   HoldingRegisters[2603] := 16#0000;
   HoldingRegisters[2604] := 16#0000;
   HoldingRegisters[2605] := 16#0000;
   HoldingRegisters[2606] := 16#0000;
   HoldingRegisters[2607] := 16#0000;
   HoldingRegisters[2608] := 16#0000;
   HoldingRegisters[2609] := 16#0000;
   HoldingRegisters[2610] := 16#0000;
   HoldingRegisters[2611] := 16#0000;
   HoldingRegisters[2612] := 16#0000;
   HoldingRegisters[2613] := 16#0000;
   HoldingRegisters[2614] := 16#0000;
   HoldingRegisters[2615] := 16#0000;
   HoldingRegisters[2616] := 16#0000;
   HoldingRegisters[2617] := 16#0000;
   HoldingRegisters[2618] := 16#0000;
   HoldingRegisters[2619] := 16#0000;
   HoldingRegisters[2620] := 16#0000;
   HoldingRegisters[2621] := 16#0000;
   HoldingRegisters[2622] := 16#0000;
   HoldingRegisters[2623] := 16#0000;
   HoldingRegisters[2624] := 16#0000;
   HoldingRegisters[2625] := 16#0000;
   HoldingRegisters[2626] := 16#0000;
   HoldingRegisters[2627] := 16#0000;
   HoldingRegisters[2628] := 16#0000;
   HoldingRegisters[2629] := 16#0000;
   HoldingRegisters[2630] := 16#0000;
   HoldingRegisters[2631] := 16#0000;
   HoldingRegisters[2632] := 16#0000;
   HoldingRegisters[2633] := 16#0000;
   HoldingRegisters[2634] := 16#0000;
   HoldingRegisters[2635] := 16#0000;
   HoldingRegisters[2636] := 16#0000;
   HoldingRegisters[2637] := 16#0000;
   HoldingRegisters[2638] := 16#0000;
   HoldingRegisters[2639] := 16#0000;
   HoldingRegisters[2640] := 16#0000;
   HoldingRegisters[2641] := 16#0000;
   HoldingRegisters[2642] := 16#0000;
   HoldingRegisters[2643] := 16#0000;
   HoldingRegisters[2644] := 16#0000;
   HoldingRegisters[2645] := 16#0000;
   HoldingRegisters[2646] := 16#0000;
   HoldingRegisters[2647] := 16#0000;
   HoldingRegisters[2648] := 16#0000;
   HoldingRegisters[2649] := 16#0000;
   HoldingRegisters[2650] := 16#0000;
   HoldingRegisters[2651] := 16#0000;
   HoldingRegisters[2652] := 16#0000;
   HoldingRegisters[2653] := 16#0000;
   HoldingRegisters[2654] := 16#0000;
   HoldingRegisters[2655] := 16#0000;
   HoldingRegisters[2656] := 16#0000;
   HoldingRegisters[2657] := 16#0000;
   HoldingRegisters[2658] := 16#0000;
   HoldingRegisters[2659] := 16#0000;
   HoldingRegisters[2660] := 16#0000;
   HoldingRegisters[2661] := 16#0000;
   HoldingRegisters[2662] := 16#0000;
   HoldingRegisters[2663] := 16#0000;
   HoldingRegisters[2664] := 16#0000;
   HoldingRegisters[2665] := 16#0000;
   HoldingRegisters[2666] := 16#0000;
   HoldingRegisters[2667] := 16#0000;
   HoldingRegisters[2668] := 16#0000;
   HoldingRegisters[2669] := 16#0000;
   HoldingRegisters[2670] := 16#0000;
   HoldingRegisters[2671] := 16#0000;
   HoldingRegisters[2672] := 16#0000;
   HoldingRegisters[2673] := 16#0000;
   HoldingRegisters[2674] := 16#0000;
   HoldingRegisters[2675] := 16#0000;
   HoldingRegisters[2676] := 16#0000;
   HoldingRegisters[2677] := 16#0000;
   HoldingRegisters[2678] := 16#0000;
   HoldingRegisters[2679] := 16#0000;
   HoldingRegisters[2680] := 16#0000;
   HoldingRegisters[2681] := 16#0000;
   HoldingRegisters[2682] := 16#0000;
   HoldingRegisters[2683] := 16#0000;
   HoldingRegisters[2684] := 16#0000;
   HoldingRegisters[2685] := 16#0000;
   HoldingRegisters[2686] := 16#0000;
   HoldingRegisters[2687] := 16#0000;
   HoldingRegisters[2688] := 16#0000;
   HoldingRegisters[2689] := 16#0000;
   HoldingRegisters[2690] := 16#0000;
   HoldingRegisters[2691] := 16#0000;
   HoldingRegisters[2692] := 16#0000;
   HoldingRegisters[2693] := 16#0000;
   HoldingRegisters[2694] := 16#0000;
   HoldingRegisters[2695] := 16#0000;
   HoldingRegisters[2696] := 16#0000;
   HoldingRegisters[2697] := 16#0000;
   HoldingRegisters[2698] := 16#0000;
   HoldingRegisters[2699] := 16#0000;
   HoldingRegisters[2700] := 16#0000;
   HoldingRegisters[2701] := 16#0000;
   HoldingRegisters[2702] := 16#0000;
   HoldingRegisters[2703] := 16#0000;
   HoldingRegisters[2704] := 16#0000;
   HoldingRegisters[2705] := 16#0000;
   HoldingRegisters[2706] := 16#0000;
   HoldingRegisters[2707] := 16#0000;
   HoldingRegisters[2708] := 16#0000;
   HoldingRegisters[2709] := 16#0000;
   HoldingRegisters[2710] := 16#0000;
   HoldingRegisters[2711] := 16#0000;
   HoldingRegisters[2712] := 16#0000;
   HoldingRegisters[2713] := 16#0000;
   HoldingRegisters[2714] := 16#0000;
   HoldingRegisters[2715] := 16#0000;
   HoldingRegisters[2716] := 16#0000;
   HoldingRegisters[2717] := 16#0000;
   HoldingRegisters[2718] := 16#0000;
   HoldingRegisters[2719] := 16#0000;
   HoldingRegisters[2720] := 16#0000;
   HoldingRegisters[2721] := 16#0000;
   HoldingRegisters[2722] := 16#0000;
   HoldingRegisters[2723] := 16#0000;
   HoldingRegisters[2724] := 16#0000;
   HoldingRegisters[2725] := 16#0000;
   HoldingRegisters[2726] := 16#0000;
   HoldingRegisters[2727] := 16#0000;
   HoldingRegisters[2728] := 16#0000;
   HoldingRegisters[2729] := 16#0000;
   HoldingRegisters[2730] := 16#0000;
   HoldingRegisters[2731] := 16#0000;
   HoldingRegisters[2732] := 16#0000;
   HoldingRegisters[2733] := 16#0000;
   HoldingRegisters[2734] := 16#0000;
   HoldingRegisters[2735] := 16#0000;
   HoldingRegisters[2736] := 16#0000;
   HoldingRegisters[2737] := 16#0000;
   HoldingRegisters[2738] := 16#0000;
   HoldingRegisters[2739] := 16#0000;
   HoldingRegisters[2740] := 16#0000;
   HoldingRegisters[2741] := 16#0000;
   HoldingRegisters[2742] := 16#0000;
   HoldingRegisters[2743] := 16#0000;
   HoldingRegisters[2744] := 16#0000;
   HoldingRegisters[2745] := 16#0000;
   HoldingRegisters[2746] := 16#0000;
   HoldingRegisters[2747] := 16#0000;
   HoldingRegisters[2748] := 16#0000;
   HoldingRegisters[2749] := 16#0000;
   HoldingRegisters[2750] := 16#0000;
   HoldingRegisters[2751] := 16#0000;
   HoldingRegisters[2752] := 16#0000;
   HoldingRegisters[2753] := 16#0000;
   HoldingRegisters[2754] := 16#0000;
   HoldingRegisters[2755] := 16#0000;
   HoldingRegisters[2756] := 16#0000;
   HoldingRegisters[2757] := 16#0000;
   HoldingRegisters[2758] := 16#0000;
   HoldingRegisters[2759] := 16#0000;
   HoldingRegisters[2760] := 16#0000;
   HoldingRegisters[2761] := 16#0000;
   HoldingRegisters[2762] := 16#0000;
   HoldingRegisters[2763] := 16#0000;
   HoldingRegisters[2764] := 16#0000;
   HoldingRegisters[2765] := 16#0000;
   HoldingRegisters[2766] := 16#0000;
   HoldingRegisters[2767] := 16#0000;
   HoldingRegisters[2768] := 16#0000;
   HoldingRegisters[2769] := 16#0000;
   HoldingRegisters[2770] := 16#0000;
   HoldingRegisters[2771] := 16#0000;
   HoldingRegisters[2772] := 16#0000;
   HoldingRegisters[2773] := 16#0000;
   HoldingRegisters[2774] := 16#0000;
   HoldingRegisters[2775] := 16#0000;
   HoldingRegisters[2776] := 16#0000;
   HoldingRegisters[2777] := 16#0000;
   HoldingRegisters[2778] := 16#0000;
   HoldingRegisters[2779] := 16#0000;
   HoldingRegisters[2780] := 16#0000;
   HoldingRegisters[2781] := 16#0000;
   HoldingRegisters[2782] := 16#0000;
   HoldingRegisters[2783] := 16#0000;
   HoldingRegisters[2784] := 16#0000;
   HoldingRegisters[2785] := 16#0000;
   HoldingRegisters[2786] := 16#0000;
   HoldingRegisters[2787] := 16#0000;
   HoldingRegisters[2788] := 16#0000;
   HoldingRegisters[2789] := 16#0000;
   HoldingRegisters[2790] := 16#0000;
   HoldingRegisters[2791] := 16#0000;
   HoldingRegisters[2792] := 16#0000;
   HoldingRegisters[2793] := 16#0000;
   HoldingRegisters[2794] := 16#0000;
   HoldingRegisters[2795] := 16#0000;
   HoldingRegisters[2796] := 16#0000;
   HoldingRegisters[2797] := 16#0000;
   HoldingRegisters[2798] := 16#0000;
   HoldingRegisters[2799] := 16#0000;
   HoldingRegisters[2800] := 16#0000;
   HoldingRegisters[2801] := 16#0000;
   HoldingRegisters[2802] := 16#0000;
   HoldingRegisters[2803] := 16#0000;
   HoldingRegisters[2804] := 16#0000;
   HoldingRegisters[2805] := 16#0000;
   HoldingRegisters[2806] := 16#0000;
   HoldingRegisters[2807] := 16#0000;
   HoldingRegisters[2808] := 16#0000;
   HoldingRegisters[2809] := 16#0000;
   HoldingRegisters[2810] := 16#0000;
   HoldingRegisters[2811] := 16#0000;
   HoldingRegisters[2812] := 16#0000;
   HoldingRegisters[2813] := 16#0000;
   HoldingRegisters[2814] := 16#0000;
   HoldingRegisters[2815] := 16#0000;
   HoldingRegisters[2816] := 16#0000;
   HoldingRegisters[2817] := 16#0000;
   HoldingRegisters[2818] := 16#0000;
   HoldingRegisters[2819] := 16#0000;
   HoldingRegisters[2820] := 16#0000;
   HoldingRegisters[2821] := 16#0000;
   HoldingRegisters[2822] := 16#0000;
   HoldingRegisters[2823] := 16#0000;
   HoldingRegisters[2824] := 16#0000;
   HoldingRegisters[2825] := 16#0000;
   HoldingRegisters[2826] := 16#0000;
   HoldingRegisters[2827] := 16#0000;
   HoldingRegisters[2828] := 16#0000;
   HoldingRegisters[2829] := 16#0000;
   HoldingRegisters[2830] := 16#0000;
   HoldingRegisters[2831] := 16#0000;
   HoldingRegisters[2832] := 16#0000;
   HoldingRegisters[2833] := 16#0000;
   HoldingRegisters[2834] := 16#0000;
   HoldingRegisters[2835] := 16#0000;
   HoldingRegisters[2836] := 16#0000;
   HoldingRegisters[2837] := 16#0000;
   HoldingRegisters[2838] := 16#0000;
   HoldingRegisters[2839] := 16#0000;
   HoldingRegisters[2840] := 16#0000;
   HoldingRegisters[2841] := 16#0000;
   HoldingRegisters[2842] := 16#0000;
   HoldingRegisters[2843] := 16#0000;
   HoldingRegisters[2844] := 16#0000;
   HoldingRegisters[2845] := 16#0000;
   HoldingRegisters[2846] := 16#0000;
   HoldingRegisters[2847] := 16#0000;
   HoldingRegisters[2848] := 16#0000;
   HoldingRegisters[2849] := 16#0000;
   HoldingRegisters[2850] := 16#0000;
   HoldingRegisters[2851] := 16#0000;
   HoldingRegisters[2852] := 16#0000;
   HoldingRegisters[2853] := 16#0000;
   HoldingRegisters[2854] := 16#0000;
   HoldingRegisters[2855] := 16#0000;
   HoldingRegisters[2856] := 16#0000;
   HoldingRegisters[2857] := 16#0000;
   HoldingRegisters[2858] := 16#0000;
   HoldingRegisters[2859] := 16#0000;
   HoldingRegisters[2860] := 16#0000;
   HoldingRegisters[2861] := 16#0000;
   HoldingRegisters[2862] := 16#0000;
   HoldingRegisters[2863] := 16#0000;
   HoldingRegisters[2864] := 16#0000;
   HoldingRegisters[2865] := 16#0000;
   HoldingRegisters[2866] := 16#0000;
   HoldingRegisters[2867] := 16#0000;
   HoldingRegisters[2868] := 16#0000;
   HoldingRegisters[2869] := 16#0000;
   HoldingRegisters[2870] := 16#0000;
   HoldingRegisters[2871] := 16#0000;
   HoldingRegisters[2872] := 16#0000;
   HoldingRegisters[2873] := 16#0000;
   HoldingRegisters[2874] := 16#0000;
   HoldingRegisters[2875] := 16#0000;
   HoldingRegisters[2876] := 16#0000;
   HoldingRegisters[2877] := 16#0000;
   HoldingRegisters[2878] := 16#0000;
   HoldingRegisters[2879] := 16#0000;
   HoldingRegisters[2880] := 16#0000;
   HoldingRegisters[2881] := 16#0000;
   HoldingRegisters[2882] := 16#0000;
   HoldingRegisters[2883] := 16#0000;
   HoldingRegisters[2884] := 16#0000;
   HoldingRegisters[2885] := 16#0000;
   HoldingRegisters[2886] := 16#0000;
   HoldingRegisters[2887] := 16#0000;
   HoldingRegisters[2888] := 16#0000;
   HoldingRegisters[2889] := 16#0000;
   HoldingRegisters[2890] := 16#0000;
   HoldingRegisters[2891] := 16#0000;
   HoldingRegisters[2892] := 16#0000;
   HoldingRegisters[2893] := 16#0000;
   HoldingRegisters[2894] := 16#0000;
   HoldingRegisters[2895] := 16#0000;
   HoldingRegisters[2896] := 16#0000;
   HoldingRegisters[2897] := 16#0000;
   HoldingRegisters[2898] := 16#0000;
   HoldingRegisters[2899] := 16#0000;
   HoldingRegisters[2900] := 16#0000;
   HoldingRegisters[2901] := 16#0000;
   HoldingRegisters[2902] := 16#0000;
   HoldingRegisters[2903] := 16#0000;
   HoldingRegisters[2904] := 16#0000;
   HoldingRegisters[2905] := 16#0000;
   HoldingRegisters[2906] := 16#0000;
   HoldingRegisters[2907] := 16#0000;
   HoldingRegisters[2908] := 16#0000;
   HoldingRegisters[2909] := 16#0000;
   HoldingRegisters[2910] := 16#0000;
   HoldingRegisters[2911] := 16#0000;
   HoldingRegisters[2912] := 16#0000;
   HoldingRegisters[2913] := 16#0000;
   HoldingRegisters[2914] := 16#0000;
   HoldingRegisters[2915] := 16#0000;
   HoldingRegisters[2916] := 16#0000;
   HoldingRegisters[2917] := 16#0000;
   HoldingRegisters[2918] := 16#0000;
   HoldingRegisters[2919] := 16#0000;
   HoldingRegisters[2920] := 16#0000;
   HoldingRegisters[2921] := 16#0000;
   HoldingRegisters[2922] := 16#0000;
   HoldingRegisters[2923] := 16#0000;
   HoldingRegisters[2924] := 16#0000;
   HoldingRegisters[2925] := 16#0000;
   HoldingRegisters[2926] := 16#0000;
   HoldingRegisters[2927] := 16#0000;
   HoldingRegisters[2928] := 16#0000;
   HoldingRegisters[2929] := 16#0000;
   HoldingRegisters[2930] := 16#0000;
   HoldingRegisters[2931] := 16#0000;
   HoldingRegisters[2932] := 16#0000;
   HoldingRegisters[2933] := 16#0000;
   HoldingRegisters[2934] := 16#0000;
   HoldingRegisters[2935] := 16#0000;
   HoldingRegisters[2936] := 16#0000;
   HoldingRegisters[2937] := 16#0000;
   HoldingRegisters[2938] := 16#0000;
   HoldingRegisters[2939] := 16#0000;
   HoldingRegisters[2940] := 16#0000;
   HoldingRegisters[2941] := 16#0000;
   HoldingRegisters[2942] := 16#0000;
   HoldingRegisters[2943] := 16#0000;
   HoldingRegisters[2944] := 16#0000;
   HoldingRegisters[2945] := 16#0000;
   HoldingRegisters[2946] := 16#0000;
   HoldingRegisters[2947] := 16#0000;
   HoldingRegisters[2948] := 16#0000;
   HoldingRegisters[2949] := 16#0000;
   HoldingRegisters[2950] := 16#0000;
   HoldingRegisters[2951] := 16#0000;
   HoldingRegisters[2952] := 16#0000;
   HoldingRegisters[2953] := 16#0000;
   HoldingRegisters[2954] := 16#0000;
   HoldingRegisters[2955] := 16#0000;
   HoldingRegisters[2956] := 16#0000;
   HoldingRegisters[2957] := 16#0000;
   HoldingRegisters[2958] := 16#0000;
   HoldingRegisters[2959] := 16#0000;
   HoldingRegisters[2960] := 16#0000;
   HoldingRegisters[2961] := 16#0000;
   HoldingRegisters[2962] := 16#0000;
   HoldingRegisters[2963] := 16#0000;
   HoldingRegisters[2964] := 16#0000;
   HoldingRegisters[2965] := 16#0000;
   HoldingRegisters[2966] := 16#0000;
   HoldingRegisters[2967] := 16#0000;
   HoldingRegisters[2968] := 16#0000;
   HoldingRegisters[2969] := 16#0000;
   HoldingRegisters[2970] := 16#0000;
   HoldingRegisters[2971] := 16#0000;
   HoldingRegisters[2972] := 16#0000;
   HoldingRegisters[2973] := 16#0000;
   HoldingRegisters[2974] := 16#0000;
   HoldingRegisters[2975] := 16#0000;
   HoldingRegisters[2976] := 16#0000;
   HoldingRegisters[2977] := 16#0000;
   HoldingRegisters[2978] := 16#0000;
   HoldingRegisters[2979] := 16#0000;
   HoldingRegisters[2980] := 16#0000;
   HoldingRegisters[2981] := 16#0000;
   HoldingRegisters[2982] := 16#0000;
   HoldingRegisters[2983] := 16#0000;
   HoldingRegisters[2984] := 16#0000;
   HoldingRegisters[2985] := 16#0000;
   HoldingRegisters[2986] := 16#0000;
   HoldingRegisters[2987] := 16#0000;
   HoldingRegisters[2988] := 16#0000;
   HoldingRegisters[2989] := 16#0000;
   HoldingRegisters[2990] := 16#0000;
   HoldingRegisters[2991] := 16#0000;
   HoldingRegisters[2992] := 16#0000;
   HoldingRegisters[2993] := 16#0000;
   HoldingRegisters[2994] := 16#0000;
   HoldingRegisters[2995] := 16#0000;
   HoldingRegisters[2996] := 16#0000;
   HoldingRegisters[2997] := 16#0000;
   HoldingRegisters[2998] := 16#0000;
   HoldingRegisters[2999] := 16#0000;
   HoldingRegisters[3000] := 16#0000;
   HoldingRegisters[3001] := 16#0000;
   HoldingRegisters[3002] := 16#0000;
   HoldingRegisters[3003] := 16#0000;
   HoldingRegisters[3004] := 16#0000;
   HoldingRegisters[3005] := 16#0000;
   HoldingRegisters[3006] := 16#0000;
   HoldingRegisters[3007] := 16#0000;
   HoldingRegisters[3008] := 16#0000;
   HoldingRegisters[3009] := 16#0000;
   HoldingRegisters[3010] := 16#0000;
   HoldingRegisters[3011] := 16#0000;
   HoldingRegisters[3012] := 16#0000;
   HoldingRegisters[3013] := 16#0000;
   HoldingRegisters[3014] := 16#0000;
   HoldingRegisters[3015] := 16#0000;
   HoldingRegisters[3016] := 16#0000;
   HoldingRegisters[3017] := 16#0000;
   HoldingRegisters[3018] := 16#0000;
   HoldingRegisters[3019] := 16#0000;
   HoldingRegisters[3020] := 16#0000;
   HoldingRegisters[3021] := 16#0000;
   HoldingRegisters[3022] := 16#0000;
   HoldingRegisters[3023] := 16#0000;
   HoldingRegisters[3024] := 16#0000;
   HoldingRegisters[3025] := 16#0000;
   HoldingRegisters[3026] := 16#0000;
   HoldingRegisters[3027] := 16#0000;
   HoldingRegisters[3028] := 16#0000;
   HoldingRegisters[3029] := 16#0000;
   HoldingRegisters[3030] := 16#0000;
   HoldingRegisters[3031] := 16#0000;
   HoldingRegisters[3032] := 16#0000;
   HoldingRegisters[3033] := 16#0000;
   HoldingRegisters[3034] := 16#0000;
   HoldingRegisters[3035] := 16#0000;
   HoldingRegisters[3036] := 16#0000;
   HoldingRegisters[3037] := 16#0000;
   HoldingRegisters[3038] := 16#0000;
   HoldingRegisters[3039] := 16#0000;
   HoldingRegisters[3040] := 16#0000;
   HoldingRegisters[3041] := 16#0000;
   HoldingRegisters[3042] := 16#0000;
   HoldingRegisters[3043] := 16#0000;
   HoldingRegisters[3044] := 16#0000;
   HoldingRegisters[3045] := 16#0000;
   HoldingRegisters[3046] := 16#0000;
   HoldingRegisters[3047] := 16#0000;
   HoldingRegisters[3048] := 16#0000;
   HoldingRegisters[3049] := 16#0000;
   HoldingRegisters[3050] := 16#0000;
   HoldingRegisters[3051] := 16#0000;
   HoldingRegisters[3052] := 16#0000;
   HoldingRegisters[3053] := 16#0000;
   HoldingRegisters[3054] := 16#0000;
   HoldingRegisters[3055] := 16#0000;
   HoldingRegisters[3056] := 16#0000;
   HoldingRegisters[3057] := 16#0000;
   HoldingRegisters[3058] := 16#0000;
   HoldingRegisters[3059] := 16#0000;
   HoldingRegisters[3060] := 16#0000;
   HoldingRegisters[3061] := 16#0000;
   HoldingRegisters[3062] := 16#0000;
   HoldingRegisters[3063] := 16#0000;
   HoldingRegisters[3064] := 16#0000;
   HoldingRegisters[3065] := 16#0000;
   HoldingRegisters[3066] := 16#0000;
   HoldingRegisters[3067] := 16#0000;
   HoldingRegisters[3068] := 16#0000;
   HoldingRegisters[3069] := 16#0000;
   HoldingRegisters[3070] := 16#0000;
   HoldingRegisters[3071] := 16#0000;
   HoldingRegisters[3072] := 16#0000;
   HoldingRegisters[3073] := 16#0000;
   HoldingRegisters[3074] := 16#0000;
   HoldingRegisters[3075] := 16#0000;
   HoldingRegisters[3076] := 16#0000;
   HoldingRegisters[3077] := 16#0000;
   HoldingRegisters[3078] := 16#0000;
   HoldingRegisters[3079] := 16#0000;
   HoldingRegisters[3080] := 16#0000;
   HoldingRegisters[3081] := 16#0000;
   HoldingRegisters[3082] := 16#0000;
   HoldingRegisters[3083] := 16#0000;
   HoldingRegisters[3084] := 16#0000;
   HoldingRegisters[3085] := 16#0000;
   HoldingRegisters[3086] := 16#0000;
   HoldingRegisters[3087] := 16#0000;
   HoldingRegisters[3088] := 16#0000;
   HoldingRegisters[3089] := 16#0000;
   HoldingRegisters[3090] := 16#0000;
   HoldingRegisters[3091] := 16#0000;
   HoldingRegisters[3092] := 16#0000;
   HoldingRegisters[3093] := 16#0000;
   HoldingRegisters[3094] := 16#0000;
   HoldingRegisters[3095] := 16#0000;
   HoldingRegisters[3096] := 16#0000;
   HoldingRegisters[3097] := 16#0000;
   HoldingRegisters[3098] := 16#0000;
   HoldingRegisters[3099] := 16#0000;
   HoldingRegisters[3100] := 16#0000;
   HoldingRegisters[3101] := 16#0000;
   HoldingRegisters[3102] := 16#0000;
   HoldingRegisters[3103] := 16#0000;
   HoldingRegisters[3104] := 16#0000;
   HoldingRegisters[3105] := 16#0000;
   HoldingRegisters[3106] := 16#0000;
   HoldingRegisters[3107] := 16#0000;
   HoldingRegisters[3108] := 16#0000;
   HoldingRegisters[3109] := 16#0000;
   HoldingRegisters[3110] := 16#0000;
   HoldingRegisters[3111] := 16#0000;
   HoldingRegisters[3112] := 16#0000;
   HoldingRegisters[3113] := 16#0000;
   HoldingRegisters[3114] := 16#0000;
   HoldingRegisters[3115] := 16#0000;
   HoldingRegisters[3116] := 16#0000;
   HoldingRegisters[3117] := 16#0000;
   HoldingRegisters[3118] := 16#0000;
   HoldingRegisters[3119] := 16#0000;
   HoldingRegisters[3120] := 16#0000;
   HoldingRegisters[3121] := 16#0000;
   HoldingRegisters[3122] := 16#0000;
   HoldingRegisters[3123] := 16#0000;
   HoldingRegisters[3124] := 16#0000;
   HoldingRegisters[3125] := 16#0000;
   HoldingRegisters[3126] := 16#0000;
   HoldingRegisters[3127] := 16#0000;
   HoldingRegisters[3128] := 16#0000;
   HoldingRegisters[3129] := 16#0000;
   HoldingRegisters[3130] := 16#0000;
   HoldingRegisters[3131] := 16#0000;
   HoldingRegisters[3132] := 16#0000;
   HoldingRegisters[3133] := 16#0000;
   HoldingRegisters[3134] := 16#0000;
   HoldingRegisters[3135] := 16#0000;
   HoldingRegisters[3136] := 16#0000;
   HoldingRegisters[3137] := 16#0000;
   HoldingRegisters[3138] := 16#0000;
   HoldingRegisters[3139] := 16#0000;
   HoldingRegisters[3140] := 16#0000;
   HoldingRegisters[3141] := 16#0000;
   HoldingRegisters[3142] := 16#0000;
   HoldingRegisters[3143] := 16#0000;
   HoldingRegisters[3144] := 16#0000;
   HoldingRegisters[3145] := 16#0000;
   HoldingRegisters[3146] := 16#0000;
   HoldingRegisters[3147] := 16#0000;
   HoldingRegisters[3148] := 16#0000;
   HoldingRegisters[3149] := 16#0000;
   HoldingRegisters[3150] := 16#0000;
   HoldingRegisters[3151] := 16#0000;
   HoldingRegisters[3152] := 16#0000;
   HoldingRegisters[3153] := 16#0000;
   HoldingRegisters[3154] := 16#0000;
   HoldingRegisters[3155] := 16#0000;
   HoldingRegisters[3156] := 16#0000;
   HoldingRegisters[3157] := 16#0000;
   HoldingRegisters[3158] := 16#0000;
   HoldingRegisters[3159] := 16#0000;
   HoldingRegisters[3160] := 16#0000;
   HoldingRegisters[3161] := 16#0000;
   HoldingRegisters[3162] := 16#0000;
   HoldingRegisters[3163] := 16#0000;
   HoldingRegisters[3164] := 16#0000;
   HoldingRegisters[3165] := 16#0000;
   HoldingRegisters[3166] := 16#0000;
   HoldingRegisters[3167] := 16#0000;
   HoldingRegisters[3168] := 16#0000;
   HoldingRegisters[3169] := 16#0000;
   HoldingRegisters[3170] := 16#0000;
   HoldingRegisters[3171] := 16#0000;
   HoldingRegisters[3172] := 16#0000;
   HoldingRegisters[3173] := 16#0000;
   HoldingRegisters[3174] := 16#0000;
   HoldingRegisters[3175] := 16#0000;
   HoldingRegisters[3176] := 16#0000;
   HoldingRegisters[3177] := 16#0000;
   HoldingRegisters[3178] := 16#0000;
   HoldingRegisters[3179] := 16#0000;
   HoldingRegisters[3180] := 16#0000;
   HoldingRegisters[3181] := 16#0000;
   HoldingRegisters[3182] := 16#0000;
   HoldingRegisters[3183] := 16#0000;
   HoldingRegisters[3184] := 16#0000;
   HoldingRegisters[3185] := 16#0000;
   HoldingRegisters[3186] := 16#0000;
   HoldingRegisters[3187] := 16#0000;
   HoldingRegisters[3188] := 16#0000;
   HoldingRegisters[3189] := 16#0000;
   HoldingRegisters[3190] := 16#0000;
   HoldingRegisters[3191] := 16#0000;
   HoldingRegisters[3192] := 16#0000;
   HoldingRegisters[3193] := 16#0000;
   HoldingRegisters[3194] := 16#0000;
   HoldingRegisters[3195] := 16#0000;
   HoldingRegisters[3196] := 16#0000;
   HoldingRegisters[3197] := 16#0000;
   HoldingRegisters[3198] := 16#0000;
   HoldingRegisters[3199] := 16#0000;
   HoldingRegisters[3200] := 16#0000;
   HoldingRegisters[3201] := 16#0000;
   HoldingRegisters[3202] := 16#0000;
   HoldingRegisters[3203] := 16#0000;
   HoldingRegisters[3204] := 16#0000;
   HoldingRegisters[3205] := 16#0000;
   HoldingRegisters[3206] := 16#0000;
   HoldingRegisters[3207] := 16#0000;
   HoldingRegisters[3208] := 16#0000;
   HoldingRegisters[3209] := 16#0000;
   HoldingRegisters[3210] := 16#0000;
   HoldingRegisters[3211] := 16#0000;
   HoldingRegisters[3212] := 16#0000;
   HoldingRegisters[3213] := 16#0000;
   HoldingRegisters[3214] := 16#0000;
   HoldingRegisters[3215] := 16#0000;
   HoldingRegisters[3216] := 16#0000;
   HoldingRegisters[3217] := 16#0000;
   HoldingRegisters[3218] := 16#0000;
   HoldingRegisters[3219] := 16#0000;
   HoldingRegisters[3220] := 16#0000;
   HoldingRegisters[3221] := 16#0000;
   HoldingRegisters[3222] := 16#0000;
   HoldingRegisters[3223] := 16#0000;
   HoldingRegisters[3224] := 16#0000;
   HoldingRegisters[3225] := 16#0000;
   HoldingRegisters[3226] := 16#0000;
   HoldingRegisters[3227] := 16#0000;
   HoldingRegisters[3228] := 16#0000;
   HoldingRegisters[3229] := 16#0000;
   HoldingRegisters[3230] := 16#0000;
   HoldingRegisters[3231] := 16#0000;
   HoldingRegisters[3232] := 16#0000;
   HoldingRegisters[3233] := 16#0000;
   HoldingRegisters[3234] := 16#0000;
   HoldingRegisters[3235] := 16#0000;
   HoldingRegisters[3236] := 16#0000;
   HoldingRegisters[3237] := 16#0000;
   HoldingRegisters[3238] := 16#0000;
   HoldingRegisters[3239] := 16#0000;
   HoldingRegisters[3240] := 16#0000;
   HoldingRegisters[3241] := 16#0000;
   HoldingRegisters[3242] := 16#0000;
   HoldingRegisters[3243] := 16#0000;
   HoldingRegisters[3244] := 16#0000;
   HoldingRegisters[3245] := 16#0000;
   HoldingRegisters[3246] := 16#0000;
   HoldingRegisters[3247] := 16#0000;
   HoldingRegisters[3248] := 16#0000;
   HoldingRegisters[3249] := 16#0000;
   HoldingRegisters[3250] := 16#0000;
   HoldingRegisters[3251] := 16#0000;
   HoldingRegisters[3252] := 16#0000;
   HoldingRegisters[3253] := 16#0000;
   HoldingRegisters[3254] := 16#0000;
   HoldingRegisters[3255] := 16#0000;
   HoldingRegisters[3256] := 16#0000;
   HoldingRegisters[3257] := 16#0000;
   HoldingRegisters[3258] := 16#0000;
   HoldingRegisters[3259] := 16#0000;
   HoldingRegisters[3260] := 16#0000;
   HoldingRegisters[3261] := 16#0000;
   HoldingRegisters[3262] := 16#0000;
   HoldingRegisters[3263] := 16#0000;
   HoldingRegisters[3264] := 16#0000;
   HoldingRegisters[3265] := 16#0000;
   HoldingRegisters[3266] := 16#0000;
   HoldingRegisters[3267] := 16#0000;
   HoldingRegisters[3268] := 16#0000;
   HoldingRegisters[3269] := 16#0000;
   HoldingRegisters[3270] := 16#0000;
   HoldingRegisters[3271] := 16#0000;
   HoldingRegisters[3272] := 16#0000;
   HoldingRegisters[3273] := 16#0000;
   HoldingRegisters[3274] := 16#0000;
   HoldingRegisters[3275] := 16#0000;
   HoldingRegisters[3276] := 16#0000;
   HoldingRegisters[3277] := 16#0000;
   HoldingRegisters[3278] := 16#0000;
   HoldingRegisters[3279] := 16#0000;
   HoldingRegisters[3280] := 16#0000;
   HoldingRegisters[3281] := 16#0000;
   HoldingRegisters[3282] := 16#0000;
   HoldingRegisters[3283] := 16#0000;
   HoldingRegisters[3284] := 16#0000;
   HoldingRegisters[3285] := 16#0000;
   HoldingRegisters[3286] := 16#0000;
   HoldingRegisters[3287] := 16#0000;
   HoldingRegisters[3288] := 16#0000;
   HoldingRegisters[3289] := 16#0000;
   HoldingRegisters[3290] := 16#0000;
   HoldingRegisters[3291] := 16#0000;
   HoldingRegisters[3292] := 16#0000;
   HoldingRegisters[3293] := 16#0000;
   HoldingRegisters[3294] := 16#0000;
   HoldingRegisters[3295] := 16#0000;
   HoldingRegisters[3296] := 16#0000;
   HoldingRegisters[3297] := 16#0000;
   HoldingRegisters[3298] := 16#0000;
   HoldingRegisters[3299] := 16#0000;
   HoldingRegisters[3300] := 16#0000;
   HoldingRegisters[3301] := 16#0000;
   HoldingRegisters[3302] := 16#0000;
   HoldingRegisters[3303] := 16#0000;
   HoldingRegisters[3304] := 16#0000;
   HoldingRegisters[3305] := 16#0000;
   HoldingRegisters[3306] := 16#0000;
   HoldingRegisters[3307] := 16#0000;
   HoldingRegisters[3308] := 16#0000;
   HoldingRegisters[3309] := 16#0000;
   HoldingRegisters[3310] := 16#0000;
   HoldingRegisters[3311] := 16#0000;
   HoldingRegisters[3312] := 16#0000;
   HoldingRegisters[3313] := 16#0000;
   HoldingRegisters[3314] := 16#0000;
   HoldingRegisters[3315] := 16#0000;
   HoldingRegisters[3316] := 16#0000;
   HoldingRegisters[3317] := 16#0000;
   HoldingRegisters[3318] := 16#0000;
   HoldingRegisters[3319] := 16#0000;
   HoldingRegisters[3320] := 16#0000;
   HoldingRegisters[3321] := 16#0000;
   HoldingRegisters[3322] := 16#0000;
   HoldingRegisters[3323] := 16#0000;
   HoldingRegisters[3324] := 16#0000;
   HoldingRegisters[3325] := 16#0000;
   HoldingRegisters[3326] := 16#0000;
   HoldingRegisters[3327] := 16#0000;
   HoldingRegisters[3328] := 16#0000;
   HoldingRegisters[3329] := 16#0000;
   HoldingRegisters[3330] := 16#0000;
   HoldingRegisters[3331] := 16#0000;
   HoldingRegisters[3332] := 16#0000;
   HoldingRegisters[3333] := 16#0000;
   HoldingRegisters[3334] := 16#0000;
   HoldingRegisters[3335] := 16#0000;
   HoldingRegisters[3336] := 16#0000;
   HoldingRegisters[3337] := 16#0000;
   HoldingRegisters[3338] := 16#0000;
   HoldingRegisters[3339] := 16#0000;
   HoldingRegisters[3340] := 16#0000;
   HoldingRegisters[3341] := 16#0000;
   HoldingRegisters[3342] := 16#0000;
   HoldingRegisters[3343] := 16#0000;
   HoldingRegisters[3344] := 16#0000;
   HoldingRegisters[3345] := 16#0000;
   HoldingRegisters[3346] := 16#0000;
   HoldingRegisters[3347] := 16#0000;
   HoldingRegisters[3348] := 16#0000;
   HoldingRegisters[3349] := 16#0000;
   HoldingRegisters[3350] := 16#0000;
   HoldingRegisters[3351] := 16#0000;
   HoldingRegisters[3352] := 16#0000;
   HoldingRegisters[3353] := 16#0000;
   HoldingRegisters[3354] := 16#0000;
   HoldingRegisters[3355] := 16#0000;
   HoldingRegisters[3356] := 16#0000;
   HoldingRegisters[3357] := 16#0000;
   HoldingRegisters[3358] := 16#0000;
   HoldingRegisters[3359] := 16#0000;
   HoldingRegisters[3360] := 16#0000;
   HoldingRegisters[3361] := 16#0000;
   HoldingRegisters[3362] := 16#0000;
   HoldingRegisters[3363] := 16#0000;
   HoldingRegisters[3364] := 16#0000;
   HoldingRegisters[3365] := 16#0000;
   HoldingRegisters[3366] := 16#0000;
   HoldingRegisters[3367] := 16#0000;
   HoldingRegisters[3368] := 16#0000;
   HoldingRegisters[3369] := 16#0000;
   HoldingRegisters[3370] := 16#0000;
   HoldingRegisters[3371] := 16#0000;
   HoldingRegisters[3372] := 16#0000;
   HoldingRegisters[3373] := 16#0000;
   HoldingRegisters[3374] := 16#0000;
   HoldingRegisters[3375] := 16#0000;
   HoldingRegisters[3376] := 16#0000;
   HoldingRegisters[3377] := 16#0000;
   HoldingRegisters[3378] := 16#0000;
   HoldingRegisters[3379] := 16#0000;
   HoldingRegisters[3380] := 16#0000;
   HoldingRegisters[3381] := 16#0000;
   HoldingRegisters[3382] := 16#0000;
   HoldingRegisters[3383] := 16#0000;
   HoldingRegisters[3384] := 16#0000;
   HoldingRegisters[3385] := 16#0000;
   HoldingRegisters[3386] := 16#0000;
   HoldingRegisters[3387] := 16#0000;
   HoldingRegisters[3388] := 16#0000;
   HoldingRegisters[3389] := 16#0000;
   HoldingRegisters[3390] := 16#0000;
   HoldingRegisters[3391] := 16#0000;
   HoldingRegisters[3392] := 16#0000;
   HoldingRegisters[3393] := 16#0000;
   HoldingRegisters[3394] := 16#0000;
   HoldingRegisters[3395] := 16#0000;
   HoldingRegisters[3396] := 16#0000;
   HoldingRegisters[3397] := 16#0000;
   HoldingRegisters[3398] := 16#0000;
   HoldingRegisters[3399] := 16#0000;
   HoldingRegisters[3400] := 16#0000;
   HoldingRegisters[3401] := 16#0000;
   HoldingRegisters[3402] := 16#0000;
   HoldingRegisters[3403] := 16#0000;
   HoldingRegisters[3404] := 16#0000;
   HoldingRegisters[3405] := 16#0000;
   HoldingRegisters[3406] := 16#0000;
   HoldingRegisters[3407] := 16#0000;
   HoldingRegisters[3408] := 16#0000;
   HoldingRegisters[3409] := 16#0000;
   HoldingRegisters[3410] := 16#0000;
   HoldingRegisters[3411] := 16#0000;
   HoldingRegisters[3412] := 16#0000;
   HoldingRegisters[3413] := 16#0000;
   HoldingRegisters[3414] := 16#0000;
   HoldingRegisters[3415] := 16#0000;
   HoldingRegisters[3416] := 16#0000;
   HoldingRegisters[3417] := 16#0000;
   HoldingRegisters[3418] := 16#0000;
   HoldingRegisters[3419] := 16#0000;
   HoldingRegisters[3420] := 16#0000;
   HoldingRegisters[3421] := 16#0000;
   HoldingRegisters[3422] := 16#0000;
   HoldingRegisters[3423] := 16#0000;
   HoldingRegisters[3424] := 16#0000;
   HoldingRegisters[3425] := 16#0000;
   HoldingRegisters[3426] := 16#0000;
   HoldingRegisters[3427] := 16#0000;
   HoldingRegisters[3428] := 16#0000;
   HoldingRegisters[3429] := 16#0000;
   HoldingRegisters[3430] := 16#0000;
   HoldingRegisters[3431] := 16#0000;
   HoldingRegisters[3432] := 16#0000;
   HoldingRegisters[3433] := 16#0000;
   HoldingRegisters[3434] := 16#0000;
   HoldingRegisters[3435] := 16#0000;
   HoldingRegisters[3436] := 16#0000;
   HoldingRegisters[3437] := 16#0000;
   HoldingRegisters[3438] := 16#0000;
   HoldingRegisters[3439] := 16#0000;
   HoldingRegisters[3440] := 16#0000;
   HoldingRegisters[3441] := 16#0000;
   HoldingRegisters[3442] := 16#0000;
   HoldingRegisters[3443] := 16#0000;
   HoldingRegisters[3444] := 16#0000;
   HoldingRegisters[3445] := 16#0000;
   HoldingRegisters[3446] := 16#0000;
   HoldingRegisters[3447] := 16#0000;
   HoldingRegisters[3448] := 16#0000;
   HoldingRegisters[3449] := 16#0000;
   HoldingRegisters[3450] := 16#0000;
   HoldingRegisters[3451] := 16#0000;
   HoldingRegisters[3452] := 16#0000;
   HoldingRegisters[3453] := 16#0000;
   HoldingRegisters[3454] := 16#0000;
   HoldingRegisters[3455] := 16#0000;
   HoldingRegisters[3456] := 16#0000;
   HoldingRegisters[3457] := 16#0000;
   HoldingRegisters[3458] := 16#0000;
   HoldingRegisters[3459] := 16#0000;
   HoldingRegisters[3460] := 16#0000;
   HoldingRegisters[3461] := 16#0000;
   HoldingRegisters[3462] := 16#0000;
   HoldingRegisters[3463] := 16#0000;
   HoldingRegisters[3464] := 16#0000;
   HoldingRegisters[3465] := 16#0000;
   HoldingRegisters[3466] := 16#0000;
   HoldingRegisters[3467] := 16#0000;
   HoldingRegisters[3468] := 16#0000;
   HoldingRegisters[3469] := 16#0000;
   HoldingRegisters[3470] := 16#0000;
   HoldingRegisters[3471] := 16#0000;
   HoldingRegisters[3472] := 16#0000;
   HoldingRegisters[3473] := 16#0000;
   HoldingRegisters[3474] := 16#0000;
   HoldingRegisters[3475] := 16#0000;
   HoldingRegisters[3476] := 16#0000;
   HoldingRegisters[3477] := 16#0000;
   HoldingRegisters[3478] := 16#0000;
   HoldingRegisters[3479] := 16#0000;
   HoldingRegisters[3480] := 16#0000;
   HoldingRegisters[3481] := 16#0000;
   HoldingRegisters[3482] := 16#0000;
   HoldingRegisters[3483] := 16#0000;
   HoldingRegisters[3484] := 16#0000;
   HoldingRegisters[3485] := 16#0000;
   HoldingRegisters[3486] := 16#0000;
   HoldingRegisters[3487] := 16#0000;
   HoldingRegisters[3488] := 16#0000;
   HoldingRegisters[3489] := 16#0000;
   HoldingRegisters[3490] := 16#0000;
   HoldingRegisters[3491] := 16#0000;
   HoldingRegisters[3492] := 16#0000;
   HoldingRegisters[3493] := 16#0000;
   HoldingRegisters[3494] := 16#0000;
   HoldingRegisters[3495] := 16#0000;
   HoldingRegisters[3496] := 16#0000;
   HoldingRegisters[3497] := 16#0000;
   HoldingRegisters[3498] := 16#0000;
   HoldingRegisters[3499] := 16#0000;
   HoldingRegisters[3500] := 16#0000;
   HoldingRegisters[3501] := 16#0000;
   HoldingRegisters[3502] := 16#0000;
   HoldingRegisters[3503] := 16#0000;
   HoldingRegisters[3504] := 16#0000;
   HoldingRegisters[3505] := 16#0000;
   HoldingRegisters[3506] := 16#0000;
   HoldingRegisters[3507] := 16#0000;
   HoldingRegisters[3508] := 16#0000;
   HoldingRegisters[3509] := 16#0000;
   HoldingRegisters[3510] := 16#0000;
   HoldingRegisters[3511] := 16#0000;
   HoldingRegisters[3512] := 16#0000;
   HoldingRegisters[3513] := 16#0000;
   HoldingRegisters[3514] := 16#0000;
   HoldingRegisters[3515] := 16#0000;
   HoldingRegisters[3516] := 16#0000;
   HoldingRegisters[3517] := 16#0000;
   HoldingRegisters[3518] := 16#0000;
   HoldingRegisters[3519] := 16#0000;
   HoldingRegisters[3520] := 16#0000;
   HoldingRegisters[3521] := 16#0000;
   HoldingRegisters[3522] := 16#0000;
   HoldingRegisters[3523] := 16#0000;
   HoldingRegisters[3524] := 16#0000;
   HoldingRegisters[3525] := 16#0000;
   HoldingRegisters[3526] := 16#0000;
   HoldingRegisters[3527] := 16#0000;
   HoldingRegisters[3528] := 16#0000;
   HoldingRegisters[3529] := 16#0000;
   HoldingRegisters[3530] := 16#0000;
   HoldingRegisters[3531] := 16#0000;
   HoldingRegisters[3532] := 16#0000;
   HoldingRegisters[3533] := 16#0000;
   HoldingRegisters[3534] := 16#0000;
   HoldingRegisters[3535] := 16#0000;
   HoldingRegisters[3536] := 16#0000;
   HoldingRegisters[3537] := 16#0000;
   HoldingRegisters[3538] := 16#0000;
   HoldingRegisters[3539] := 16#0000;
   HoldingRegisters[3540] := 16#0000;
   HoldingRegisters[3541] := 16#0000;
   HoldingRegisters[3542] := 16#0000;
   HoldingRegisters[3543] := 16#0000;
   HoldingRegisters[3544] := 16#0000;
   HoldingRegisters[3545] := 16#0000;
   HoldingRegisters[3546] := 16#0000;
   HoldingRegisters[3547] := 16#0000;
   HoldingRegisters[3548] := 16#0000;
   HoldingRegisters[3549] := 16#0000;
   HoldingRegisters[3550] := 16#0000;
   HoldingRegisters[3551] := 16#0000;
   HoldingRegisters[3552] := 16#0000;
   HoldingRegisters[3553] := 16#0000;
   HoldingRegisters[3554] := 16#0000;
   HoldingRegisters[3555] := 16#0000;
   HoldingRegisters[3556] := 16#0000;
   HoldingRegisters[3557] := 16#0000;
   HoldingRegisters[3558] := 16#0000;
   HoldingRegisters[3559] := 16#0000;
   HoldingRegisters[3560] := 16#0000;
   HoldingRegisters[3561] := 16#0000;
   HoldingRegisters[3562] := 16#0000;
   HoldingRegisters[3563] := 16#0000;
   HoldingRegisters[3564] := 16#0000;
   HoldingRegisters[3565] := 16#0000;
   HoldingRegisters[3566] := 16#0000;
   HoldingRegisters[3567] := 16#0000;
   HoldingRegisters[3568] := 16#0000;
   HoldingRegisters[3569] := 16#0000;
   HoldingRegisters[3570] := 16#0000;
   HoldingRegisters[3571] := 16#0000;
   HoldingRegisters[3572] := 16#0000;
   HoldingRegisters[3573] := 16#0000;
   HoldingRegisters[3574] := 16#0000;
   HoldingRegisters[3575] := 16#0000;
   HoldingRegisters[3576] := 16#0000;
   HoldingRegisters[3577] := 16#0000;
   HoldingRegisters[3578] := 16#0000;
   HoldingRegisters[3579] := 16#0000;
   HoldingRegisters[3580] := 16#0000;
   HoldingRegisters[3581] := 16#0000;
   HoldingRegisters[3582] := 16#0000;
   HoldingRegisters[3583] := 16#0000;
   HoldingRegisters[3584] := 16#0000;
   HoldingRegisters[3585] := 16#0000;
   HoldingRegisters[3586] := 16#0000;
   HoldingRegisters[3587] := 16#0000;
   HoldingRegisters[3588] := 16#0000;
   HoldingRegisters[3589] := 16#0000;
   HoldingRegisters[3590] := 16#0000;
   HoldingRegisters[3591] := 16#0000;
   HoldingRegisters[3592] := 16#0000;
   HoldingRegisters[3593] := 16#0000;
   HoldingRegisters[3594] := 16#0000;
   HoldingRegisters[3595] := 16#0000;
   HoldingRegisters[3596] := 16#0000;
   HoldingRegisters[3597] := 16#0000;
   HoldingRegisters[3598] := 16#0000;
   HoldingRegisters[3599] := 16#0000;
   HoldingRegisters[3600] := 16#0000;
   HoldingRegisters[3601] := 16#0000;
   HoldingRegisters[3602] := 16#0000;
   HoldingRegisters[3603] := 16#0000;
   HoldingRegisters[3604] := 16#0000;
   HoldingRegisters[3605] := 16#0000;
   HoldingRegisters[3606] := 16#0000;
   HoldingRegisters[3607] := 16#0000;
   HoldingRegisters[3608] := 16#0000;
   HoldingRegisters[3609] := 16#0000;
   HoldingRegisters[3610] := 16#0000;
   HoldingRegisters[3611] := 16#0000;
   HoldingRegisters[3612] := 16#0000;
   HoldingRegisters[3613] := 16#0000;
   HoldingRegisters[3614] := 16#0000;
   HoldingRegisters[3615] := 16#0000;
   HoldingRegisters[3616] := 16#0000;
   HoldingRegisters[3617] := 16#0000;
   HoldingRegisters[3618] := 16#0000;
   HoldingRegisters[3619] := 16#0000;
   HoldingRegisters[3620] := 16#0000;
   HoldingRegisters[3621] := 16#0000;
   HoldingRegisters[3622] := 16#0000;
   HoldingRegisters[3623] := 16#0000;
   HoldingRegisters[3624] := 16#0000;
   HoldingRegisters[3625] := 16#0000;
   HoldingRegisters[3626] := 16#0000;
   HoldingRegisters[3627] := 16#0000;
   HoldingRegisters[3628] := 16#0000;
   HoldingRegisters[3629] := 16#0000;
   HoldingRegisters[3630] := 16#0000;
   HoldingRegisters[3631] := 16#0000;
   HoldingRegisters[3632] := 16#0000;
   HoldingRegisters[3633] := 16#0000;
   HoldingRegisters[3634] := 16#0000;
   HoldingRegisters[3635] := 16#0000;
   HoldingRegisters[3636] := 16#0000;
   HoldingRegisters[3637] := 16#0000;
   HoldingRegisters[3638] := 16#0000;
   HoldingRegisters[3639] := 16#0000;
   HoldingRegisters[3640] := 16#0000;
   HoldingRegisters[3641] := 16#0000;
   HoldingRegisters[3642] := 16#0000;
   HoldingRegisters[3643] := 16#0000;
   HoldingRegisters[3644] := 16#0000;
   HoldingRegisters[3645] := 16#0000;
   HoldingRegisters[3646] := 16#0000;
   HoldingRegisters[3647] := 16#0000;
   HoldingRegisters[3648] := 16#0000;
   HoldingRegisters[3649] := 16#0000;
   HoldingRegisters[3650] := 16#0000;
   HoldingRegisters[3651] := 16#0000;
   HoldingRegisters[3652] := 16#0000;
   HoldingRegisters[3653] := 16#0000;
   HoldingRegisters[3654] := 16#0000;
   HoldingRegisters[3655] := 16#0000;
   HoldingRegisters[3656] := 16#0000;
   HoldingRegisters[3657] := 16#0000;
   HoldingRegisters[3658] := 16#0000;
   HoldingRegisters[3659] := 16#0000;
   HoldingRegisters[3660] := 16#0000;
   HoldingRegisters[3661] := 16#0000;
   HoldingRegisters[3662] := 16#0000;
   HoldingRegisters[3663] := 16#0000;
   HoldingRegisters[3664] := 16#0000;
   HoldingRegisters[3665] := 16#0000;
   HoldingRegisters[3666] := 16#0000;
   HoldingRegisters[3667] := 16#0000;
   HoldingRegisters[3668] := 16#0000;
   HoldingRegisters[3669] := 16#0000;
   HoldingRegisters[3670] := 16#0000;
   HoldingRegisters[3671] := 16#0000;
   HoldingRegisters[3672] := 16#0000;
   HoldingRegisters[3673] := 16#0000;
   HoldingRegisters[3674] := 16#0000;
   HoldingRegisters[3675] := 16#0000;
   HoldingRegisters[3676] := 16#0000;
   HoldingRegisters[3677] := 16#0000;
   HoldingRegisters[3678] := 16#0000;
   HoldingRegisters[3679] := 16#0000;
   HoldingRegisters[3680] := 16#0000;
   HoldingRegisters[3681] := 16#0000;
   HoldingRegisters[3682] := 16#0000;
   HoldingRegisters[3683] := 16#0000;
   HoldingRegisters[3684] := 16#0000;
   HoldingRegisters[3685] := 16#0000;
   HoldingRegisters[3686] := 16#0000;
   HoldingRegisters[3687] := 16#0000;
   HoldingRegisters[3688] := 16#0000;
   HoldingRegisters[3689] := 16#0000;
   HoldingRegisters[3690] := 16#0000;
   HoldingRegisters[3691] := 16#0000;
   HoldingRegisters[3692] := 16#0000;
   HoldingRegisters[3693] := 16#0000;
   HoldingRegisters[3694] := 16#0000;
   HoldingRegisters[3695] := 16#0000;
   HoldingRegisters[3696] := 16#0000;
   HoldingRegisters[3697] := 16#0000;
   HoldingRegisters[3698] := 16#0000;
   HoldingRegisters[3699] := 16#0000;
   HoldingRegisters[3700] := 16#0000;
   HoldingRegisters[3701] := 16#0000;
   HoldingRegisters[3702] := 16#0000;
   HoldingRegisters[3703] := 16#0000;
   HoldingRegisters[3704] := 16#0000;
   HoldingRegisters[3705] := 16#0000;
   HoldingRegisters[3706] := 16#0000;
   HoldingRegisters[3707] := 16#0000;
   HoldingRegisters[3708] := 16#0000;
   HoldingRegisters[3709] := 16#0000;
   HoldingRegisters[3710] := 16#0000;
   HoldingRegisters[3711] := 16#0000;
   HoldingRegisters[3712] := 16#0000;
   HoldingRegisters[3713] := 16#0000;
   HoldingRegisters[3714] := 16#0000;
   HoldingRegisters[3715] := 16#0000;
   HoldingRegisters[3716] := 16#0000;
   HoldingRegisters[3717] := 16#0000;
   HoldingRegisters[3718] := 16#0000;
   HoldingRegisters[3719] := 16#0000;
   HoldingRegisters[3720] := 16#0000;
   HoldingRegisters[3721] := 16#0000;
   HoldingRegisters[3722] := 16#0000;
   HoldingRegisters[3723] := 16#0000;
   HoldingRegisters[3724] := 16#0000;
   HoldingRegisters[3725] := 16#0000;
   HoldingRegisters[3726] := 16#0000;
   HoldingRegisters[3727] := 16#0000;
   HoldingRegisters[3728] := 16#0000;
   HoldingRegisters[3729] := 16#0000;
   HoldingRegisters[3730] := 16#0000;
   HoldingRegisters[3731] := 16#0000;
   HoldingRegisters[3732] := 16#0000;
   HoldingRegisters[3733] := 16#0000;
   HoldingRegisters[3734] := 16#0000;
   HoldingRegisters[3735] := 16#0000;
   HoldingRegisters[3736] := 16#0000;
   HoldingRegisters[3737] := 16#0000;
   HoldingRegisters[3738] := 16#0000;
   HoldingRegisters[3739] := 16#0000;
   HoldingRegisters[3740] := 16#0000;
   HoldingRegisters[3741] := 16#0000;
   HoldingRegisters[3742] := 16#0000;
   HoldingRegisters[3743] := 16#0000;
   HoldingRegisters[3744] := 16#0000;
   HoldingRegisters[3745] := 16#0000;
   HoldingRegisters[3746] := 16#0000;
   HoldingRegisters[3747] := 16#0000;
   HoldingRegisters[3748] := 16#0000;
   HoldingRegisters[3749] := 16#0000;
   HoldingRegisters[3750] := 16#0000;
   HoldingRegisters[3751] := 16#0000;
   HoldingRegisters[3752] := 16#0000;
   HoldingRegisters[3753] := 16#0000;
   HoldingRegisters[3754] := 16#0000;
   HoldingRegisters[3755] := 16#0000;
   HoldingRegisters[3756] := 16#0000;
   HoldingRegisters[3757] := 16#0000;
   HoldingRegisters[3758] := 16#0000;
   HoldingRegisters[3759] := 16#0000;
   HoldingRegisters[3760] := 16#0000;
   HoldingRegisters[3761] := 16#0000;
   HoldingRegisters[3762] := 16#0000;
   HoldingRegisters[3763] := 16#0000;
   HoldingRegisters[3764] := 16#0000;
   HoldingRegisters[3765] := 16#0000;
   HoldingRegisters[3766] := 16#0000;
   HoldingRegisters[3767] := 16#0000;
   HoldingRegisters[3768] := 16#0000;
   HoldingRegisters[3769] := 16#0000;
   HoldingRegisters[3770] := 16#0000;
   HoldingRegisters[3771] := 16#0000;
   HoldingRegisters[3772] := 16#0000;
   HoldingRegisters[3773] := 16#0000;
   HoldingRegisters[3774] := 16#0000;
   HoldingRegisters[3775] := 16#0000;
   HoldingRegisters[3776] := 16#0000;
   HoldingRegisters[3777] := 16#0000;
   HoldingRegisters[3778] := 16#0000;
   HoldingRegisters[3779] := 16#0000;
   HoldingRegisters[3780] := 16#0000;
   HoldingRegisters[3781] := 16#0000;
   HoldingRegisters[3782] := 16#0000;
   HoldingRegisters[3783] := 16#0000;
   HoldingRegisters[3784] := 16#0000;
   HoldingRegisters[3785] := 16#0000;
   HoldingRegisters[3786] := 16#0000;
   HoldingRegisters[3787] := 16#0000;
   HoldingRegisters[3788] := 16#0000;
   HoldingRegisters[3789] := 16#0000;
   HoldingRegisters[3790] := 16#0000;
   HoldingRegisters[3791] := 16#0000;
   HoldingRegisters[3792] := 16#0000;
   HoldingRegisters[3793] := 16#0000;
   HoldingRegisters[3794] := 16#0000;
   HoldingRegisters[3795] := 16#0000;
   HoldingRegisters[3796] := 16#0000;
   HoldingRegisters[3797] := 16#0000;
   HoldingRegisters[3798] := 16#0000;
   HoldingRegisters[3799] := 16#0000;
   HoldingRegisters[3800] := 16#0000;
   HoldingRegisters[3801] := 16#0000;
   HoldingRegisters[3802] := 16#0000;
   HoldingRegisters[3803] := 16#0000;
   HoldingRegisters[3804] := 16#0000;
   HoldingRegisters[3805] := 16#0000;
   HoldingRegisters[3806] := 16#0000;
   HoldingRegisters[3807] := 16#0000;
   HoldingRegisters[3808] := 16#0000;
   HoldingRegisters[3809] := 16#0000;
   HoldingRegisters[3810] := 16#0000;
   HoldingRegisters[3811] := 16#0000;
   HoldingRegisters[3812] := 16#0000;
   HoldingRegisters[3813] := 16#0000;
   HoldingRegisters[3814] := 16#0000;
   HoldingRegisters[3815] := 16#0000;
   HoldingRegisters[3816] := 16#0000;
   HoldingRegisters[3817] := 16#0000;
   HoldingRegisters[3818] := 16#0000;
   HoldingRegisters[3819] := 16#0000;
   HoldingRegisters[3820] := 16#0000;
   HoldingRegisters[3821] := 16#0000;
   HoldingRegisters[3822] := 16#0000;
   HoldingRegisters[3823] := 16#0000;
   HoldingRegisters[3824] := 16#0000;
   HoldingRegisters[3825] := 16#0000;
   HoldingRegisters[3826] := 16#0000;
   HoldingRegisters[3827] := 16#0000;
   HoldingRegisters[3828] := 16#0000;
   HoldingRegisters[3829] := 16#0000;
   HoldingRegisters[3830] := 16#0000;
   HoldingRegisters[3831] := 16#0000;
   HoldingRegisters[3832] := 16#0000;
   HoldingRegisters[3833] := 16#0000;
   HoldingRegisters[3834] := 16#0000;
   HoldingRegisters[3835] := 16#0000;
   HoldingRegisters[3836] := 16#0000;
   HoldingRegisters[3837] := 16#0000;
   HoldingRegisters[3838] := 16#0000;
   HoldingRegisters[3839] := 16#0000;
   HoldingRegisters[3840] := 16#0000;
   HoldingRegisters[3841] := 16#0000;
   HoldingRegisters[3842] := 16#0000;
   HoldingRegisters[3843] := 16#0000;
   HoldingRegisters[3844] := 16#0000;
   HoldingRegisters[3845] := 16#0000;
   HoldingRegisters[3846] := 16#0000;
   HoldingRegisters[3847] := 16#0000;
   HoldingRegisters[3848] := 16#0000;
   HoldingRegisters[3849] := 16#0000;
   HoldingRegisters[3850] := 16#0000;
   HoldingRegisters[3851] := 16#0000;
   HoldingRegisters[3852] := 16#0000;
   HoldingRegisters[3853] := 16#0000;
   HoldingRegisters[3854] := 16#0000;
   HoldingRegisters[3855] := 16#0000;
   HoldingRegisters[3856] := 16#0000;
   HoldingRegisters[3857] := 16#0000;
   HoldingRegisters[3858] := 16#0000;
   HoldingRegisters[3859] := 16#0000;
   HoldingRegisters[3860] := 16#0000;
   HoldingRegisters[3861] := 16#0000;
   HoldingRegisters[3862] := 16#0000;
   HoldingRegisters[3863] := 16#0000;
   HoldingRegisters[3864] := 16#0000;
   HoldingRegisters[3865] := 16#0000;
   HoldingRegisters[3866] := 16#0000;
   HoldingRegisters[3867] := 16#0000;
   HoldingRegisters[3868] := 16#0000;
   HoldingRegisters[3869] := 16#0000;
   HoldingRegisters[3870] := 16#0000;
   HoldingRegisters[3871] := 16#0000;
   HoldingRegisters[3872] := 16#0000;
   HoldingRegisters[3873] := 16#0000;
   HoldingRegisters[3874] := 16#0000;
   HoldingRegisters[3875] := 16#0000;
   HoldingRegisters[3876] := 16#0000;
   HoldingRegisters[3877] := 16#0000;
   HoldingRegisters[3878] := 16#0000;
   HoldingRegisters[3879] := 16#0000;
   HoldingRegisters[3880] := 16#0000;
   HoldingRegisters[3881] := 16#0000;
   HoldingRegisters[3882] := 16#0000;
   HoldingRegisters[3883] := 16#0000;
   HoldingRegisters[3884] := 16#0000;
   HoldingRegisters[3885] := 16#0000;
   HoldingRegisters[3886] := 16#0000;
   HoldingRegisters[3887] := 16#0000;
   HoldingRegisters[3888] := 16#0000;
   HoldingRegisters[3889] := 16#0000;
   HoldingRegisters[3890] := 16#0000;
   HoldingRegisters[3891] := 16#0000;
   HoldingRegisters[3892] := 16#0000;
   HoldingRegisters[3893] := 16#0000;
   HoldingRegisters[3894] := 16#0000;
   HoldingRegisters[3895] := 16#0000;
   HoldingRegisters[3896] := 16#0000;
   HoldingRegisters[3897] := 16#0000;
   HoldingRegisters[3898] := 16#0000;
   HoldingRegisters[3899] := 16#0000;
   HoldingRegisters[3900] := 16#0000;
   HoldingRegisters[3901] := 16#0000;
   HoldingRegisters[3902] := 16#0000;
   HoldingRegisters[3903] := 16#0000;
   HoldingRegisters[3904] := 16#0000;
   HoldingRegisters[3905] := 16#0000;
   HoldingRegisters[3906] := 16#0000;
   HoldingRegisters[3907] := 16#0000;
   HoldingRegisters[3908] := 16#0000;
   HoldingRegisters[3909] := 16#0000;
   HoldingRegisters[3910] := 16#0000;
   HoldingRegisters[3911] := 16#0000;
   HoldingRegisters[3912] := 16#0000;
   HoldingRegisters[3913] := 16#0000;
   HoldingRegisters[3914] := 16#0000;
   HoldingRegisters[3915] := 16#0000;
   HoldingRegisters[3916] := 16#0000;
   HoldingRegisters[3917] := 16#0000;
   HoldingRegisters[3918] := 16#0000;
   HoldingRegisters[3919] := 16#0000;
   HoldingRegisters[3920] := 16#0000;
   HoldingRegisters[3921] := 16#0000;
   HoldingRegisters[3922] := 16#0000;
   HoldingRegisters[3923] := 16#0000;
   HoldingRegisters[3924] := 16#0000;
   HoldingRegisters[3925] := 16#0000;
   HoldingRegisters[3926] := 16#0000;
   HoldingRegisters[3927] := 16#0000;
   HoldingRegisters[3928] := 16#0000;
   HoldingRegisters[3929] := 16#0000;
   HoldingRegisters[3930] := 16#0000;
   HoldingRegisters[3931] := 16#0000;
   HoldingRegisters[3932] := 16#0000;
   HoldingRegisters[3933] := 16#0000;
   HoldingRegisters[3934] := 16#0000;
   HoldingRegisters[3935] := 16#0000;
   HoldingRegisters[3936] := 16#0000;
   HoldingRegisters[3937] := 16#0000;
   HoldingRegisters[3938] := 16#0000;
   HoldingRegisters[3939] := 16#0000;
   HoldingRegisters[3940] := 16#0000;
   HoldingRegisters[3941] := 16#0000;
   HoldingRegisters[3942] := 16#0000;
   HoldingRegisters[3943] := 16#0000;
   HoldingRegisters[3944] := 16#0000;
   HoldingRegisters[3945] := 16#0000;
   HoldingRegisters[3946] := 16#0000;
   HoldingRegisters[3947] := 16#0000;
   HoldingRegisters[3948] := 16#0000;
   HoldingRegisters[3949] := 16#0000;
   HoldingRegisters[3950] := 16#0000;
   HoldingRegisters[3951] := 16#0000;
   HoldingRegisters[3952] := 16#0000;
   HoldingRegisters[3953] := 16#0000;
   HoldingRegisters[3954] := 16#0000;
   HoldingRegisters[3955] := 16#0000;
   HoldingRegisters[3956] := 16#0000;
   HoldingRegisters[3957] := 16#0000;
   HoldingRegisters[3958] := 16#0000;
   HoldingRegisters[3959] := 16#0000;
   HoldingRegisters[3960] := 16#0000;
   HoldingRegisters[3961] := 16#0000;
   HoldingRegisters[3962] := 16#0000;
   HoldingRegisters[3963] := 16#0000;
   HoldingRegisters[3964] := 16#0000;
   HoldingRegisters[3965] := 16#0000;
   HoldingRegisters[3966] := 16#0000;
   HoldingRegisters[3967] := 16#0000;
   HoldingRegisters[3968] := 16#0000;
   HoldingRegisters[3969] := 16#0000;
   HoldingRegisters[3970] := 16#0000;
   HoldingRegisters[3971] := 16#0000;
   HoldingRegisters[3972] := 16#0000;
   HoldingRegisters[3973] := 16#0000;
   HoldingRegisters[3974] := 16#0000;
   HoldingRegisters[3975] := 16#0000;
   HoldingRegisters[3976] := 16#0000;
   HoldingRegisters[3977] := 16#0000;
   HoldingRegisters[3978] := 16#0000;
   HoldingRegisters[3979] := 16#0000;
   HoldingRegisters[3980] := 16#0000;
   HoldingRegisters[3981] := 16#0000;
   HoldingRegisters[3982] := 16#0000;
   HoldingRegisters[3983] := 16#0000;
   HoldingRegisters[3984] := 16#0000;
   HoldingRegisters[3985] := 16#0000;
   HoldingRegisters[3986] := 16#0000;
   HoldingRegisters[3987] := 16#0000;
   HoldingRegisters[3988] := 16#0000;
   HoldingRegisters[3989] := 16#0000;
   HoldingRegisters[3990] := 16#0000;
   HoldingRegisters[3991] := 16#0000;
   HoldingRegisters[3992] := 16#0000;
   HoldingRegisters[3993] := 16#0000;
   HoldingRegisters[3994] := 16#0000;
   HoldingRegisters[3995] := 16#0000;
   HoldingRegisters[3996] := 16#0000;
   HoldingRegisters[3997] := 16#0000;
   HoldingRegisters[3998] := 16#0000;
   HoldingRegisters[3999] := 16#0000;
   HoldingRegisters[4000] := 16#0000;
   HoldingRegisters[4001] := 16#0000;
   HoldingRegisters[4002] := 16#0000;
   HoldingRegisters[4003] := 16#0000;
   HoldingRegisters[4004] := 16#0000;
   HoldingRegisters[4005] := 16#0000;
   HoldingRegisters[4006] := 16#0000;
   HoldingRegisters[4007] := 16#0000;
   HoldingRegisters[4008] := 16#0000;
   HoldingRegisters[4009] := 16#0000;
   HoldingRegisters[4010] := 16#0000;
   HoldingRegisters[4011] := 16#0000;
   HoldingRegisters[4012] := 16#0000;
   HoldingRegisters[4013] := 16#0000;
   HoldingRegisters[4014] := 16#0000;
   HoldingRegisters[4015] := 16#0000;
   HoldingRegisters[4016] := 16#0000;
   HoldingRegisters[4017] := 16#0000;
   HoldingRegisters[4018] := 16#0000;
   HoldingRegisters[4019] := 16#0000;
   HoldingRegisters[4020] := 16#0000;
   HoldingRegisters[4021] := 16#0000;
   HoldingRegisters[4022] := 16#0000;
   HoldingRegisters[4023] := 16#0000;
   HoldingRegisters[4024] := 16#0000;
   HoldingRegisters[4025] := 16#0000;
   HoldingRegisters[4026] := 16#0000;
   HoldingRegisters[4027] := 16#0000;
   HoldingRegisters[4028] := 16#0000;
   HoldingRegisters[4029] := 16#0000;
   HoldingRegisters[4030] := 16#0000;
   HoldingRegisters[4031] := 16#0000;
   HoldingRegisters[4032] := 16#0000;
   HoldingRegisters[4033] := 16#0000;
   HoldingRegisters[4034] := 16#0000;
   HoldingRegisters[4035] := 16#0000;
   HoldingRegisters[4036] := 16#0000;
   HoldingRegisters[4037] := 16#0000;
   HoldingRegisters[4038] := 16#0000;
   HoldingRegisters[4039] := 16#0000;
   HoldingRegisters[4040] := 16#0000;
   HoldingRegisters[4041] := 16#0000;
   HoldingRegisters[4042] := 16#0000;
   HoldingRegisters[4043] := 16#0000;
   HoldingRegisters[4044] := 16#0000;
   HoldingRegisters[4045] := 16#0000;
   HoldingRegisters[4046] := 16#0000;
   HoldingRegisters[4047] := 16#0000;
   HoldingRegisters[4048] := 16#0000;
   HoldingRegisters[4049] := 16#0000;
   HoldingRegisters[4050] := 16#0000;
   HoldingRegisters[4051] := 16#0000;
   HoldingRegisters[4052] := 16#0000;
   HoldingRegisters[4053] := 16#0000;
   HoldingRegisters[4054] := 16#0000;
   HoldingRegisters[4055] := 16#0000;
   HoldingRegisters[4056] := 16#0000;
   HoldingRegisters[4057] := 16#0000;
   HoldingRegisters[4058] := 16#0000;
   HoldingRegisters[4059] := 16#0000;
   HoldingRegisters[4060] := 16#0000;
   HoldingRegisters[4061] := 16#0000;
   HoldingRegisters[4062] := 16#0000;
   HoldingRegisters[4063] := 16#0000;
   HoldingRegisters[4064] := 16#0000;
   HoldingRegisters[4065] := 16#0000;
   HoldingRegisters[4066] := 16#0000;
   HoldingRegisters[4067] := 16#0000;
   HoldingRegisters[4068] := 16#0000;
   HoldingRegisters[4069] := 16#0000;
   HoldingRegisters[4070] := 16#0000;
   HoldingRegisters[4071] := 16#0000;
   HoldingRegisters[4072] := 16#0000;
   HoldingRegisters[4073] := 16#0000;
   HoldingRegisters[4074] := 16#0000;
   HoldingRegisters[4075] := 16#0000;
   HoldingRegisters[4076] := 16#0000;
   HoldingRegisters[4077] := 16#0000;
   HoldingRegisters[4078] := 16#0000;
   HoldingRegisters[4079] := 16#0000;
   HoldingRegisters[4080] := 16#0000;
   HoldingRegisters[4081] := 16#0000;
   HoldingRegisters[4082] := 16#0000;
   HoldingRegisters[4083] := 16#0000;
   HoldingRegisters[4084] := 16#0000;
   HoldingRegisters[4085] := 16#0000;
   HoldingRegisters[4086] := 16#0000;
   HoldingRegisters[4087] := 16#0000;
   HoldingRegisters[4088] := 16#0000;
   HoldingRegisters[4089] := 16#0000;
   HoldingRegisters[4090] := 16#0000;
   HoldingRegisters[4091] := 16#0000;
   HoldingRegisters[4092] := 16#0000;
   HoldingRegisters[4093] := 16#0000;
   HoldingRegisters[4094] := 16#0000;
   HoldingRegisters[4095] := 16#0000;
   HoldingRegisters[4096] := 16#0000;
   HoldingRegisters[4097] := 16#0000;
   HoldingRegisters[4098] := 16#0000;
   HoldingRegisters[4099] := 16#0000;
   HoldingRegisters[4100] := 16#0000;
   HoldingRegisters[4101] := 16#0000;
   HoldingRegisters[4102] := 16#0000;
   HoldingRegisters[4103] := 16#0000;
   HoldingRegisters[4104] := 16#0000;
   HoldingRegisters[4105] := 16#0000;
   HoldingRegisters[4106] := 16#0000;
   HoldingRegisters[4107] := 16#0000;
   HoldingRegisters[4108] := 16#0000;
   HoldingRegisters[4109] := 16#0000;
   HoldingRegisters[4110] := 16#0000;
   HoldingRegisters[4111] := 16#0000;
   HoldingRegisters[4112] := 16#0000;
   HoldingRegisters[4113] := 16#0000;
   HoldingRegisters[4114] := 16#0000;
   HoldingRegisters[4115] := 16#0000;
   HoldingRegisters[4116] := 16#0000;
   HoldingRegisters[4117] := 16#0000;
   HoldingRegisters[4118] := 16#0000;
   HoldingRegisters[4119] := 16#0000;
   HoldingRegisters[4120] := 16#0000;
   HoldingRegisters[4121] := 16#0000;
   HoldingRegisters[4122] := 16#0000;
   HoldingRegisters[4123] := 16#0000;
   HoldingRegisters[4124] := 16#0000;
   HoldingRegisters[4125] := 16#0000;
   HoldingRegisters[4126] := 16#0000;
   HoldingRegisters[4127] := 16#0000;
   HoldingRegisters[4128] := 16#0000;
   HoldingRegisters[4129] := 16#0000;
   HoldingRegisters[4130] := 16#0000;
   HoldingRegisters[4131] := 16#0000;
   HoldingRegisters[4132] := 16#0000;
   HoldingRegisters[4133] := 16#0000;
   HoldingRegisters[4134] := 16#0000;
   HoldingRegisters[4135] := 16#0000;
   HoldingRegisters[4136] := 16#0000;
   HoldingRegisters[4137] := 16#0000;
   HoldingRegisters[4138] := 16#0000;
   HoldingRegisters[4139] := 16#0000;
   HoldingRegisters[4140] := 16#0000;
   HoldingRegisters[4141] := 16#0000;
   HoldingRegisters[4142] := 16#0000;
   HoldingRegisters[4143] := 16#0000;
   HoldingRegisters[4144] := 16#0000;
   HoldingRegisters[4145] := 16#0000;
   HoldingRegisters[4146] := 16#0000;
   HoldingRegisters[4147] := 16#0000;
   HoldingRegisters[4148] := 16#0000;
   HoldingRegisters[4149] := 16#0000;
   HoldingRegisters[4150] := 16#0000;
   HoldingRegisters[4151] := 16#0000;
   HoldingRegisters[4152] := 16#0000;
   HoldingRegisters[4153] := 16#0000;
   HoldingRegisters[4154] := 16#0000;
   HoldingRegisters[4155] := 16#0000;
   HoldingRegisters[4156] := 16#0000;
   HoldingRegisters[4157] := 16#0000;
   HoldingRegisters[4158] := 16#0000;
   HoldingRegisters[4159] := 16#0000;
   HoldingRegisters[4160] := 16#0000;
   HoldingRegisters[4161] := 16#0000;
   HoldingRegisters[4162] := 16#0000;
   HoldingRegisters[4163] := 16#0000;
   HoldingRegisters[4164] := 16#0000;
   HoldingRegisters[4165] := 16#0000;
   HoldingRegisters[4166] := 16#0000;
   HoldingRegisters[4167] := 16#0000;
   HoldingRegisters[4168] := 16#0000;
   HoldingRegisters[4169] := 16#0000;
   HoldingRegisters[4170] := 16#0000;
   HoldingRegisters[4171] := 16#0000;
   HoldingRegisters[4172] := 16#0000;
   HoldingRegisters[4173] := 16#0000;
   HoldingRegisters[4174] := 16#0000;
   HoldingRegisters[4175] := 16#0000;
   HoldingRegisters[4176] := 16#0000;
   HoldingRegisters[4177] := 16#0000;
   HoldingRegisters[4178] := 16#0000;
   HoldingRegisters[4179] := 16#0000;
   HoldingRegisters[4180] := 16#0000;
   HoldingRegisters[4181] := 16#0000;
   HoldingRegisters[4182] := 16#0000;
   HoldingRegisters[4183] := 16#0000;
   HoldingRegisters[4184] := 16#0000;
   HoldingRegisters[4185] := 16#0000;
   HoldingRegisters[4186] := 16#0000;
   HoldingRegisters[4187] := 16#0000;
   HoldingRegisters[4188] := 16#0000;
   HoldingRegisters[4189] := 16#0000;
   HoldingRegisters[4190] := 16#0000;
   HoldingRegisters[4191] := 16#0000;
   HoldingRegisters[4192] := 16#0000;
   HoldingRegisters[4193] := 16#0000;
   HoldingRegisters[4194] := 16#0000;
   HoldingRegisters[4195] := 16#0000;
   HoldingRegisters[4196] := 16#0000;
   HoldingRegisters[4197] := 16#0000;
   HoldingRegisters[4198] := 16#0000;
   HoldingRegisters[4199] := 16#0000;
   HoldingRegisters[4200] := 16#0000;
   HoldingRegisters[4201] := 16#0000;
   HoldingRegisters[4202] := 16#0000;
   HoldingRegisters[4203] := 16#0000;
   HoldingRegisters[4204] := 16#0000;
   HoldingRegisters[4205] := 16#0000;
   HoldingRegisters[4206] := 16#0000;
   HoldingRegisters[4207] := 16#0000;
   HoldingRegisters[4208] := 16#0000;
   HoldingRegisters[4209] := 16#0000;
   HoldingRegisters[4210] := 16#0000;
   HoldingRegisters[4211] := 16#0000;
   HoldingRegisters[4212] := 16#0000;
   HoldingRegisters[4213] := 16#0000;
   HoldingRegisters[4214] := 16#0000;
   HoldingRegisters[4215] := 16#0000;
   HoldingRegisters[4216] := 16#0000;
   HoldingRegisters[4217] := 16#0000;
   HoldingRegisters[4218] := 16#0000;
   HoldingRegisters[4219] := 16#0000;
   HoldingRegisters[4220] := 16#0000;
   HoldingRegisters[4221] := 16#0000;
   HoldingRegisters[4222] := 16#0000;
   HoldingRegisters[4223] := 16#0000;
   HoldingRegisters[4224] := 16#0000;
   HoldingRegisters[4225] := 16#0000;
   HoldingRegisters[4226] := 16#0000;
   HoldingRegisters[4227] := 16#0000;
   HoldingRegisters[4228] := 16#0000;
   HoldingRegisters[4229] := 16#0000;
   HoldingRegisters[4230] := 16#0000;
   HoldingRegisters[4231] := 16#0000;
   HoldingRegisters[4232] := 16#0000;
   HoldingRegisters[4233] := 16#0000;
   HoldingRegisters[4234] := 16#0000;
   HoldingRegisters[4235] := 16#0000;
   HoldingRegisters[4236] := 16#0000;
   HoldingRegisters[4237] := 16#0000;
   HoldingRegisters[4238] := 16#0000;
   HoldingRegisters[4239] := 16#0000;
   HoldingRegisters[4240] := 16#0000;
   HoldingRegisters[4241] := 16#0000;
   HoldingRegisters[4242] := 16#0000;
   HoldingRegisters[4243] := 16#0000;
   HoldingRegisters[4244] := 16#0000;
   HoldingRegisters[4245] := 16#0000;
   HoldingRegisters[4246] := 16#0000;
   HoldingRegisters[4247] := 16#0000;
   HoldingRegisters[4248] := 16#0000;
   HoldingRegisters[4249] := 16#0000;
   HoldingRegisters[4250] := 16#0000;
   HoldingRegisters[4251] := 16#0000;
   HoldingRegisters[4252] := 16#0000;
   HoldingRegisters[4253] := 16#0000;
   HoldingRegisters[4254] := 16#0000;
   HoldingRegisters[4255] := 16#0000;
   HoldingRegisters[4256] := 16#0000;
   HoldingRegisters[4257] := 16#0000;
   HoldingRegisters[4258] := 16#0000;
   HoldingRegisters[4259] := 16#0000;
   HoldingRegisters[4260] := 16#0000;
   HoldingRegisters[4261] := 16#0000;
   HoldingRegisters[4262] := 16#0000;
   HoldingRegisters[4263] := 16#0000;
   HoldingRegisters[4264] := 16#0000;
   HoldingRegisters[4265] := 16#0000;
   HoldingRegisters[4266] := 16#0000;
   HoldingRegisters[4267] := 16#0000;
   HoldingRegisters[4268] := 16#0000;
   HoldingRegisters[4269] := 16#0000;
   HoldingRegisters[4270] := 16#0000;
   HoldingRegisters[4271] := 16#0000;
   HoldingRegisters[4272] := 16#0000;
   HoldingRegisters[4273] := 16#0000;
   HoldingRegisters[4274] := 16#0000;
   HoldingRegisters[4275] := 16#0000;
   HoldingRegisters[4276] := 16#0000;
   HoldingRegisters[4277] := 16#0000;
   HoldingRegisters[4278] := 16#0000;
   HoldingRegisters[4279] := 16#0000;
   HoldingRegisters[4280] := 16#0000;
   HoldingRegisters[4281] := 16#0000;
   HoldingRegisters[4282] := 16#0000;
   HoldingRegisters[4283] := 16#0000;
   HoldingRegisters[4284] := 16#0000;
   HoldingRegisters[4285] := 16#0000;
   HoldingRegisters[4286] := 16#0000;
   HoldingRegisters[4287] := 16#0000;
   HoldingRegisters[4288] := 16#0000;
   HoldingRegisters[4289] := 16#0000;
   HoldingRegisters[4290] := 16#0000;
   HoldingRegisters[4291] := 16#0000;
   HoldingRegisters[4292] := 16#0000;
   HoldingRegisters[4293] := 16#0000;
   HoldingRegisters[4294] := 16#0000;
   HoldingRegisters[4295] := 16#0000;
   HoldingRegisters[4296] := 16#0000;
   HoldingRegisters[4297] := 16#0000;
   HoldingRegisters[4298] := 16#0000;
   HoldingRegisters[4299] := 16#0000;
   HoldingRegisters[4300] := 16#0000;
   HoldingRegisters[4301] := 16#0000;
   HoldingRegisters[4302] := 16#0000;
   HoldingRegisters[4303] := 16#0000;
   HoldingRegisters[4304] := 16#0000;
   HoldingRegisters[4305] := 16#0000;
   HoldingRegisters[4306] := 16#0000;
   HoldingRegisters[4307] := 16#0000;
   HoldingRegisters[4308] := 16#0000;
   HoldingRegisters[4309] := 16#0000;
   HoldingRegisters[4310] := 16#0000;
   HoldingRegisters[4311] := 16#0000;
   HoldingRegisters[4312] := 16#0000;
   HoldingRegisters[4313] := 16#0000;
   HoldingRegisters[4314] := 16#0000;
   HoldingRegisters[4315] := 16#0000;
   HoldingRegisters[4316] := 16#0000;
   HoldingRegisters[4317] := 16#0000;
   HoldingRegisters[4318] := 16#0000;
   HoldingRegisters[4319] := 16#0000;
   HoldingRegisters[4320] := 16#0000;
   HoldingRegisters[4321] := 16#0000;
   HoldingRegisters[4322] := 16#0000;
   HoldingRegisters[4323] := 16#0000;
   HoldingRegisters[4324] := 16#0000;
   HoldingRegisters[4325] := 16#0000;
   HoldingRegisters[4326] := 16#0000;
   HoldingRegisters[4327] := 16#0000;
   HoldingRegisters[4328] := 16#0000;
   HoldingRegisters[4329] := 16#0000;
   HoldingRegisters[4330] := 16#0000;
   HoldingRegisters[4331] := 16#0000;
   HoldingRegisters[4332] := 16#0000;
   HoldingRegisters[4333] := 16#0000;
   HoldingRegisters[4334] := 16#0000;
   HoldingRegisters[4335] := 16#0000;
   HoldingRegisters[4336] := 16#0000;
   HoldingRegisters[4337] := 16#0000;
   HoldingRegisters[4338] := 16#0000;
   HoldingRegisters[4339] := 16#0000;
   HoldingRegisters[4340] := 16#0000;
   HoldingRegisters[4341] := 16#0000;
   HoldingRegisters[4342] := 16#0000;
   HoldingRegisters[4343] := 16#0000;
   HoldingRegisters[4344] := 16#0000;
   HoldingRegisters[4345] := 16#0000;
   HoldingRegisters[4346] := 16#0000;
   HoldingRegisters[4347] := 16#0000;
   HoldingRegisters[4348] := 16#0000;
   HoldingRegisters[4349] := 16#0000;
   HoldingRegisters[4350] := 16#0000;
   HoldingRegisters[4351] := 16#0000;
   HoldingRegisters[4352] := 16#0000;
   HoldingRegisters[4353] := 16#0000;
   HoldingRegisters[4354] := 16#0000;
   HoldingRegisters[4355] := 16#0000;
   HoldingRegisters[4356] := 16#0000;
   HoldingRegisters[4357] := 16#0000;
   HoldingRegisters[4358] := 16#0000;
   HoldingRegisters[4359] := 16#0000;
   HoldingRegisters[4360] := 16#0000;
   HoldingRegisters[4361] := 16#0000;
   HoldingRegisters[4362] := 16#0000;
   HoldingRegisters[4363] := 16#0000;
   HoldingRegisters[4364] := 16#0000;
   HoldingRegisters[4365] := 16#0000;
   HoldingRegisters[4366] := 16#0000;
   HoldingRegisters[4367] := 16#0000;
   HoldingRegisters[4368] := 16#0000;
   HoldingRegisters[4369] := 16#0000;
   HoldingRegisters[4370] := 16#0000;
   HoldingRegisters[4371] := 16#0000;
   HoldingRegisters[4372] := 16#0000;
   HoldingRegisters[4373] := 16#0000;
   HoldingRegisters[4374] := 16#0000;
   HoldingRegisters[4375] := 16#0000;
   HoldingRegisters[4376] := 16#0000;
   HoldingRegisters[4377] := 16#0000;
   HoldingRegisters[4378] := 16#0000;
   HoldingRegisters[4379] := 16#0000;
   HoldingRegisters[4380] := 16#0000;
   HoldingRegisters[4381] := 16#0000;
   HoldingRegisters[4382] := 16#0000;
   HoldingRegisters[4383] := 16#0000;
   HoldingRegisters[4384] := 16#0000;
   HoldingRegisters[4385] := 16#0000;
   HoldingRegisters[4386] := 16#0000;
   HoldingRegisters[4387] := 16#0000;
   HoldingRegisters[4388] := 16#0000;
   HoldingRegisters[4389] := 16#0000;
   HoldingRegisters[4390] := 16#0000;
   HoldingRegisters[4391] := 16#0000;
   HoldingRegisters[4392] := 16#0000;
   HoldingRegisters[4393] := 16#0000;
   HoldingRegisters[4394] := 16#0000;
   HoldingRegisters[4395] := 16#0000;
   HoldingRegisters[4396] := 16#0000;
   HoldingRegisters[4397] := 16#0000;
   HoldingRegisters[4398] := 16#0000;
   HoldingRegisters[4399] := 16#0000;
   HoldingRegisters[4400] := 16#0000;
   HoldingRegisters[4401] := 16#0000;
   HoldingRegisters[4402] := 16#0000;
   HoldingRegisters[4403] := 16#0000;
   HoldingRegisters[4404] := 16#0000;
   HoldingRegisters[4405] := 16#0000;
   HoldingRegisters[4406] := 16#0000;
   HoldingRegisters[4407] := 16#0000;
   HoldingRegisters[4408] := 16#0000;
   HoldingRegisters[4409] := 16#0000;
   HoldingRegisters[4410] := 16#0000;
   HoldingRegisters[4411] := 16#0000;
   HoldingRegisters[4412] := 16#0000;
   HoldingRegisters[4413] := 16#0000;
   HoldingRegisters[4414] := 16#0000;
   HoldingRegisters[4415] := 16#0000;
   HoldingRegisters[4416] := 16#0000;
   HoldingRegisters[4417] := 16#0000;
   HoldingRegisters[4418] := 16#0000;
   HoldingRegisters[4419] := 16#0000;
   HoldingRegisters[4420] := 16#0000;
   HoldingRegisters[4421] := 16#0000;
   HoldingRegisters[4422] := 16#0000;
   HoldingRegisters[4423] := 16#0000;
   HoldingRegisters[4424] := 16#0000;
   HoldingRegisters[4425] := 16#0000;
   HoldingRegisters[4426] := 16#0000;
   HoldingRegisters[4427] := 16#0000;
   HoldingRegisters[4428] := 16#0000;
   HoldingRegisters[4429] := 16#0000;
   HoldingRegisters[4430] := 16#0000;
   HoldingRegisters[4431] := 16#0000;
   HoldingRegisters[4432] := 16#0000;
   HoldingRegisters[4433] := 16#0000;
   HoldingRegisters[4434] := 16#0000;
   HoldingRegisters[4435] := 16#0000;
   HoldingRegisters[4436] := 16#0000;
   HoldingRegisters[4437] := 16#0000;
   HoldingRegisters[4438] := 16#0000;
   HoldingRegisters[4439] := 16#0000;
   HoldingRegisters[4440] := 16#0000;
   HoldingRegisters[4441] := 16#0000;
   HoldingRegisters[4442] := 16#0000;
   HoldingRegisters[4443] := 16#0000;
   HoldingRegisters[4444] := 16#0000;
   HoldingRegisters[4445] := 16#0000;
   HoldingRegisters[4446] := 16#0000;
   HoldingRegisters[4447] := 16#0000;
   HoldingRegisters[4448] := 16#0000;
   HoldingRegisters[4449] := 16#0000;
   HoldingRegisters[4450] := 16#0000;
   HoldingRegisters[4451] := 16#0000;
   HoldingRegisters[4452] := 16#0000;
   HoldingRegisters[4453] := 16#0000;
   HoldingRegisters[4454] := 16#0000;
   HoldingRegisters[4455] := 16#0000;
   HoldingRegisters[4456] := 16#0000;
   HoldingRegisters[4457] := 16#0000;
   HoldingRegisters[4458] := 16#0000;
   HoldingRegisters[4459] := 16#0000;
   HoldingRegisters[4460] := 16#0000;
   HoldingRegisters[4461] := 16#0000;
   HoldingRegisters[4462] := 16#0000;
   HoldingRegisters[4463] := 16#0000;
   HoldingRegisters[4464] := 16#0000;
   HoldingRegisters[4465] := 16#0000;
   HoldingRegisters[4466] := 16#0000;
   HoldingRegisters[4467] := 16#0000;
   HoldingRegisters[4468] := 16#0000;
   HoldingRegisters[4469] := 16#0000;
   HoldingRegisters[4470] := 16#0000;
   HoldingRegisters[4471] := 16#0000;
   HoldingRegisters[4472] := 16#0000;
   HoldingRegisters[4473] := 16#0000;
   HoldingRegisters[4474] := 16#0000;
   HoldingRegisters[4475] := 16#0000;
   HoldingRegisters[4476] := 16#0000;
   HoldingRegisters[4477] := 16#0000;
   HoldingRegisters[4478] := 16#0000;
   HoldingRegisters[4479] := 16#0000;
   HoldingRegisters[4480] := 16#0000;
   HoldingRegisters[4481] := 16#0000;
   HoldingRegisters[4482] := 16#0000;
   HoldingRegisters[4483] := 16#0000;
   HoldingRegisters[4484] := 16#0000;
   HoldingRegisters[4485] := 16#0000;
   HoldingRegisters[4486] := 16#0000;
   HoldingRegisters[4487] := 16#0000;
   HoldingRegisters[4488] := 16#0000;
   HoldingRegisters[4489] := 16#0000;
   HoldingRegisters[4490] := 16#0000;
   HoldingRegisters[4491] := 16#0000;
   HoldingRegisters[4492] := 16#0000;
   HoldingRegisters[4493] := 16#0000;
   HoldingRegisters[4494] := 16#0000;
   HoldingRegisters[4495] := 16#0000;
   HoldingRegisters[4496] := 16#0000;
   HoldingRegisters[4497] := 16#0000;
   HoldingRegisters[4498] := 16#0000;
   HoldingRegisters[4499] := 16#0000;
   HoldingRegisters[4500] := 16#0000;
   HoldingRegisters[4501] := 16#0000;
   HoldingRegisters[4502] := 16#0000;
   HoldingRegisters[4503] := 16#0000;
   HoldingRegisters[4504] := 16#0000;
   HoldingRegisters[4505] := 16#0000;
   HoldingRegisters[4506] := 16#0000;
   HoldingRegisters[4507] := 16#0000;
   HoldingRegisters[4508] := 16#0000;
   HoldingRegisters[4509] := 16#0000;
   HoldingRegisters[4510] := 16#0000;
   HoldingRegisters[4511] := 16#0000;
   HoldingRegisters[4512] := 16#0000;
   HoldingRegisters[4513] := 16#0000;
   HoldingRegisters[4514] := 16#0000;
   HoldingRegisters[4515] := 16#0000;
   HoldingRegisters[4516] := 16#0000;
   HoldingRegisters[4517] := 16#0000;
   HoldingRegisters[4518] := 16#0000;
   HoldingRegisters[4519] := 16#0000;
   HoldingRegisters[4520] := 16#0000;
   HoldingRegisters[4521] := 16#0000;
   HoldingRegisters[4522] := 16#0000;
   HoldingRegisters[4523] := 16#0000;
   HoldingRegisters[4524] := 16#0000;
   HoldingRegisters[4525] := 16#0000;
   HoldingRegisters[4526] := 16#0000;
   HoldingRegisters[4527] := 16#0000;
   HoldingRegisters[4528] := 16#0000;
   HoldingRegisters[4529] := 16#0000;
   HoldingRegisters[4530] := 16#0000;
   HoldingRegisters[4531] := 16#0000;
   HoldingRegisters[4532] := 16#0000;
   HoldingRegisters[4533] := 16#0000;
   HoldingRegisters[4534] := 16#0000;
   HoldingRegisters[4535] := 16#0000;
   HoldingRegisters[4536] := 16#0000;
   HoldingRegisters[4537] := 16#0000;
   HoldingRegisters[4538] := 16#0000;
   HoldingRegisters[4539] := 16#0000;
   HoldingRegisters[4540] := 16#0000;
   HoldingRegisters[4541] := 16#0000;
   HoldingRegisters[4542] := 16#0000;
   HoldingRegisters[4543] := 16#0000;
   HoldingRegisters[4544] := 16#0000;
   HoldingRegisters[4545] := 16#0000;
   HoldingRegisters[4546] := 16#0000;
   HoldingRegisters[4547] := 16#0000;
   HoldingRegisters[4548] := 16#0000;
   HoldingRegisters[4549] := 16#0000;
   HoldingRegisters[4550] := 16#0000;
   HoldingRegisters[4551] := 16#0000;
   HoldingRegisters[4552] := 16#0000;
   HoldingRegisters[4553] := 16#0000;
   HoldingRegisters[4554] := 16#0000;
   HoldingRegisters[4555] := 16#0000;
   HoldingRegisters[4556] := 16#0000;
   HoldingRegisters[4557] := 16#0000;
   HoldingRegisters[4558] := 16#0000;
   HoldingRegisters[4559] := 16#0000;
   HoldingRegisters[4560] := 16#0000;
   HoldingRegisters[4561] := 16#0000;
   HoldingRegisters[4562] := 16#0000;
   HoldingRegisters[4563] := 16#0000;
   HoldingRegisters[4564] := 16#0000;
   HoldingRegisters[4565] := 16#0000;
   HoldingRegisters[4566] := 16#0000;
   HoldingRegisters[4567] := 16#0000;
   HoldingRegisters[4568] := 16#0000;
   HoldingRegisters[4569] := 16#0000;
   HoldingRegisters[4570] := 16#0000;
   HoldingRegisters[4571] := 16#0000;
   HoldingRegisters[4572] := 16#0000;
   HoldingRegisters[4573] := 16#0000;
   HoldingRegisters[4574] := 16#0000;
   HoldingRegisters[4575] := 16#0000;
   HoldingRegisters[4576] := 16#0000;
   HoldingRegisters[4577] := 16#0000;
   HoldingRegisters[4578] := 16#0000;
   HoldingRegisters[4579] := 16#0000;
   HoldingRegisters[4580] := 16#0000;
   HoldingRegisters[4581] := 16#0000;
   HoldingRegisters[4582] := 16#0000;
   HoldingRegisters[4583] := 16#0000;
   HoldingRegisters[4584] := 16#0000;
   HoldingRegisters[4585] := 16#0000;
   HoldingRegisters[4586] := 16#0000;
   HoldingRegisters[4587] := 16#0000;
   HoldingRegisters[4588] := 16#0000;
   HoldingRegisters[4589] := 16#0000;
   HoldingRegisters[4590] := 16#0000;
   HoldingRegisters[4591] := 16#0000;
   HoldingRegisters[4592] := 16#0000;
   HoldingRegisters[4593] := 16#0000;
   HoldingRegisters[4594] := 16#0000;
   HoldingRegisters[4595] := 16#0000;
   HoldingRegisters[4596] := 16#0000;
   HoldingRegisters[4597] := 16#0000;
   HoldingRegisters[4598] := 16#0000;
   HoldingRegisters[4599] := 16#0000;
   HoldingRegisters[4600] := 16#0000;
   HoldingRegisters[4601] := 16#0000;
   HoldingRegisters[4602] := 16#0000;
   HoldingRegisters[4603] := 16#0000;
   HoldingRegisters[4604] := 16#0000;
   HoldingRegisters[4605] := 16#0000;
   HoldingRegisters[4606] := 16#0000;
   HoldingRegisters[4607] := 16#0000;
   HoldingRegisters[4608] := 16#0000;
   HoldingRegisters[4609] := 16#0000;
   HoldingRegisters[4610] := 16#0000;
   HoldingRegisters[4611] := 16#0000;
   HoldingRegisters[4612] := 16#0000;
   HoldingRegisters[4613] := 16#0000;
   HoldingRegisters[4614] := 16#0000;
   HoldingRegisters[4615] := 16#0000;
   HoldingRegisters[4616] := 16#0000;
   HoldingRegisters[4617] := 16#0000;
   HoldingRegisters[4618] := 16#0000;
   HoldingRegisters[4619] := 16#0000;
   HoldingRegisters[4620] := 16#0000;
   HoldingRegisters[4621] := 16#0000;
   HoldingRegisters[4622] := 16#0000;
   HoldingRegisters[4623] := 16#0000;
   HoldingRegisters[4624] := 16#0000;
   HoldingRegisters[4625] := 16#0000;
   HoldingRegisters[4626] := 16#0000;
   HoldingRegisters[4627] := 16#0000;
   HoldingRegisters[4628] := 16#0000;
   HoldingRegisters[4629] := 16#0000;
   HoldingRegisters[4630] := 16#0000;
   HoldingRegisters[4631] := 16#0000;
   HoldingRegisters[4632] := 16#0000;
   HoldingRegisters[4633] := 16#0000;
   HoldingRegisters[4634] := 16#0000;
   HoldingRegisters[4635] := 16#0000;
   HoldingRegisters[4636] := 16#0000;
   HoldingRegisters[4637] := 16#0000;
   HoldingRegisters[4638] := 16#0000;
   HoldingRegisters[4639] := 16#0000;
   HoldingRegisters[4640] := 16#0000;
   HoldingRegisters[4641] := 16#0000;
   HoldingRegisters[4642] := 16#0000;
   HoldingRegisters[4643] := 16#0000;
   HoldingRegisters[4644] := 16#0000;
   HoldingRegisters[4645] := 16#0000;
   HoldingRegisters[4646] := 16#0000;
   HoldingRegisters[4647] := 16#0000;
   HoldingRegisters[4648] := 16#0000;
   HoldingRegisters[4649] := 16#0000;
   HoldingRegisters[4650] := 16#0000;
   HoldingRegisters[4651] := 16#0000;
   HoldingRegisters[4652] := 16#0000;
   HoldingRegisters[4653] := 16#0000;
   HoldingRegisters[4654] := 16#0000;
   HoldingRegisters[4655] := 16#0000;
   HoldingRegisters[4656] := 16#0000;
   HoldingRegisters[4657] := 16#0000;
   HoldingRegisters[4658] := 16#0000;
   HoldingRegisters[4659] := 16#0000;
   HoldingRegisters[4660] := 16#0000;
   HoldingRegisters[4661] := 16#0000;
   HoldingRegisters[4662] := 16#0000;
   HoldingRegisters[4663] := 16#0000;
   HoldingRegisters[4664] := 16#0000;
   HoldingRegisters[4665] := 16#0000;
   HoldingRegisters[4666] := 16#0000;
   HoldingRegisters[4667] := 16#0000;
   HoldingRegisters[4668] := 16#0000;
   HoldingRegisters[4669] := 16#0000;
   HoldingRegisters[4670] := 16#0000;
   HoldingRegisters[4671] := 16#0000;
   HoldingRegisters[4672] := 16#0000;
   HoldingRegisters[4673] := 16#0000;
   HoldingRegisters[4674] := 16#0000;
   HoldingRegisters[4675] := 16#0000;
   HoldingRegisters[4676] := 16#0000;
   HoldingRegisters[4677] := 16#0000;
   HoldingRegisters[4678] := 16#0000;
   HoldingRegisters[4679] := 16#0000;
   HoldingRegisters[4680] := 16#0000;
   HoldingRegisters[4681] := 16#0000;
   HoldingRegisters[4682] := 16#0000;
   HoldingRegisters[4683] := 16#0000;
   HoldingRegisters[4684] := 16#0000;
   HoldingRegisters[4685] := 16#0000;
   HoldingRegisters[4686] := 16#0000;
   HoldingRegisters[4687] := 16#0000;
   HoldingRegisters[4688] := 16#0000;
   HoldingRegisters[4689] := 16#0000;
   HoldingRegisters[4690] := 16#0000;
   HoldingRegisters[4691] := 16#0000;
   HoldingRegisters[4692] := 16#0000;
   HoldingRegisters[4693] := 16#0000;
   HoldingRegisters[4694] := 16#0000;
   HoldingRegisters[4695] := 16#0000;
   HoldingRegisters[4696] := 16#0000;
   HoldingRegisters[4697] := 16#0000;
   HoldingRegisters[4698] := 16#0000;
   HoldingRegisters[4699] := 16#0000;
   HoldingRegisters[4700] := 16#0000;
   HoldingRegisters[4701] := 16#0000;
   HoldingRegisters[4702] := 16#0000;
   HoldingRegisters[4703] := 16#0000;
   HoldingRegisters[4704] := 16#0000;
   HoldingRegisters[4705] := 16#0000;
   HoldingRegisters[4706] := 16#0000;
   HoldingRegisters[4707] := 16#0000;
   HoldingRegisters[4708] := 16#0000;
   HoldingRegisters[4709] := 16#0000;
   HoldingRegisters[4710] := 16#0000;
   HoldingRegisters[4711] := 16#0000;
   HoldingRegisters[4712] := 16#0000;
   HoldingRegisters[4713] := 16#0000;
   HoldingRegisters[4714] := 16#0000;
   HoldingRegisters[4715] := 16#0000;
   HoldingRegisters[4716] := 16#0000;
   HoldingRegisters[4717] := 16#0000;
   HoldingRegisters[4718] := 16#0000;
   HoldingRegisters[4719] := 16#0000;
   HoldingRegisters[4720] := 16#0000;
   HoldingRegisters[4721] := 16#0000;
   HoldingRegisters[4722] := 16#0000;
   HoldingRegisters[4723] := 16#0000;
   HoldingRegisters[4724] := 16#0000;
   HoldingRegisters[4725] := 16#0000;
   HoldingRegisters[4726] := 16#0000;
   HoldingRegisters[4727] := 16#0000;
   HoldingRegisters[4728] := 16#0000;
   HoldingRegisters[4729] := 16#0000;
   HoldingRegisters[4730] := 16#0000;
   HoldingRegisters[4731] := 16#0000;
   HoldingRegisters[4732] := 16#0000;
   HoldingRegisters[4733] := 16#0000;
   HoldingRegisters[4734] := 16#0000;
   HoldingRegisters[4735] := 16#0000;
   HoldingRegisters[4736] := 16#0000;
   HoldingRegisters[4737] := 16#0000;
   HoldingRegisters[4738] := 16#0000;
   HoldingRegisters[4739] := 16#0000;
   HoldingRegisters[4740] := 16#0000;
   HoldingRegisters[4741] := 16#0000;
   HoldingRegisters[4742] := 16#0000;
   HoldingRegisters[4743] := 16#0000;
   HoldingRegisters[4744] := 16#0000;
   HoldingRegisters[4745] := 16#0000;
   HoldingRegisters[4746] := 16#0000;
   HoldingRegisters[4747] := 16#0000;
   HoldingRegisters[4748] := 16#0000;
   HoldingRegisters[4749] := 16#0000;
   HoldingRegisters[4750] := 16#0000;
   HoldingRegisters[4751] := 16#0000;
   HoldingRegisters[4752] := 16#0000;
   HoldingRegisters[4753] := 16#0000;
   HoldingRegisters[4754] := 16#0000;
   HoldingRegisters[4755] := 16#0000;
   HoldingRegisters[4756] := 16#0000;
   HoldingRegisters[4757] := 16#0000;
   HoldingRegisters[4758] := 16#0000;
   HoldingRegisters[4759] := 16#0000;
   HoldingRegisters[4760] := 16#0000;
   HoldingRegisters[4761] := 16#0000;
   HoldingRegisters[4762] := 16#0000;
   HoldingRegisters[4763] := 16#0000;
   HoldingRegisters[4764] := 16#0000;
   HoldingRegisters[4765] := 16#0000;
   HoldingRegisters[4766] := 16#0000;
   HoldingRegisters[4767] := 16#0000;
   HoldingRegisters[4768] := 16#0000;
   HoldingRegisters[4769] := 16#0000;
   HoldingRegisters[4770] := 16#0000;
   HoldingRegisters[4771] := 16#0000;
   HoldingRegisters[4772] := 16#0000;
   HoldingRegisters[4773] := 16#0000;
   HoldingRegisters[4774] := 16#0000;
   HoldingRegisters[4775] := 16#0000;
   HoldingRegisters[4776] := 16#0000;
   HoldingRegisters[4777] := 16#0000;
   HoldingRegisters[4778] := 16#0000;
   HoldingRegisters[4779] := 16#0000;
   HoldingRegisters[4780] := 16#0000;
   HoldingRegisters[4781] := 16#0000;
   HoldingRegisters[4782] := 16#0000;
   HoldingRegisters[4783] := 16#0000;
   HoldingRegisters[4784] := 16#0000;
   HoldingRegisters[4785] := 16#0000;
   HoldingRegisters[4786] := 16#0000;
   HoldingRegisters[4787] := 16#0000;
   HoldingRegisters[4788] := 16#0000;
   HoldingRegisters[4789] := 16#0000;
   HoldingRegisters[4790] := 16#0000;
   HoldingRegisters[4791] := 16#0000;
   HoldingRegisters[4792] := 16#0000;
   HoldingRegisters[4793] := 16#0000;
   HoldingRegisters[4794] := 16#0000;
   HoldingRegisters[4795] := 16#0000;
   HoldingRegisters[4796] := 16#0000;
   HoldingRegisters[4797] := 16#0000;
   HoldingRegisters[4798] := 16#0000;
   HoldingRegisters[4799] := 16#0000;
   HoldingRegisters[4800] := 16#0000;
   HoldingRegisters[4801] := 16#0000;
   HoldingRegisters[4802] := 16#0000;
   HoldingRegisters[4803] := 16#0000;
   HoldingRegisters[4804] := 16#0000;
   HoldingRegisters[4805] := 16#0000;
   HoldingRegisters[4806] := 16#0000;
   HoldingRegisters[4807] := 16#0000;
   HoldingRegisters[4808] := 16#0000;
   HoldingRegisters[4809] := 16#0000;
   HoldingRegisters[4810] := 16#0000;
   HoldingRegisters[4811] := 16#0000;
   HoldingRegisters[4812] := 16#0000;
   HoldingRegisters[4813] := 16#0000;
   HoldingRegisters[4814] := 16#0000;
   HoldingRegisters[4815] := 16#0000;
   HoldingRegisters[4816] := 16#0000;
   HoldingRegisters[4817] := 16#0000;
   HoldingRegisters[4818] := 16#0000;
   HoldingRegisters[4819] := 16#0000;
   HoldingRegisters[4820] := 16#0000;
   HoldingRegisters[4821] := 16#0000;
   HoldingRegisters[4822] := 16#0000;
   HoldingRegisters[4823] := 16#0000;
   HoldingRegisters[4824] := 16#0000;
   HoldingRegisters[4825] := 16#0000;
   HoldingRegisters[4826] := 16#0000;
   HoldingRegisters[4827] := 16#0000;
   HoldingRegisters[4828] := 16#0000;
   HoldingRegisters[4829] := 16#0000;
   HoldingRegisters[4830] := 16#0000;
   HoldingRegisters[4831] := 16#0000;
   HoldingRegisters[4832] := 16#0000;
   HoldingRegisters[4833] := 16#0000;
   HoldingRegisters[4834] := 16#0000;
   HoldingRegisters[4835] := 16#0000;
   HoldingRegisters[4836] := 16#0000;
   HoldingRegisters[4837] := 16#0000;
   HoldingRegisters[4838] := 16#0000;
   HoldingRegisters[4839] := 16#0000;
   HoldingRegisters[4840] := 16#0000;
   HoldingRegisters[4841] := 16#0000;
   HoldingRegisters[4842] := 16#0000;
   HoldingRegisters[4843] := 16#0000;
   HoldingRegisters[4844] := 16#0000;
   HoldingRegisters[4845] := 16#0000;
   HoldingRegisters[4846] := 16#0000;
   HoldingRegisters[4847] := 16#0000;
   HoldingRegisters[4848] := 16#0000;
   HoldingRegisters[4849] := 16#0000;
   HoldingRegisters[4850] := 16#0000;
   HoldingRegisters[4851] := 16#0000;
   HoldingRegisters[4852] := 16#0000;
   HoldingRegisters[4853] := 16#0000;
   HoldingRegisters[4854] := 16#0000;
   HoldingRegisters[4855] := 16#0000;
   HoldingRegisters[4856] := 16#0000;
   HoldingRegisters[4857] := 16#0000;
   HoldingRegisters[4858] := 16#0000;
   HoldingRegisters[4859] := 16#0000;
   HoldingRegisters[4860] := 16#0000;
   HoldingRegisters[4861] := 16#0000;
   HoldingRegisters[4862] := 16#0000;
   HoldingRegisters[4863] := 16#0000;
   HoldingRegisters[4864] := 16#0000;
   HoldingRegisters[4865] := 16#0000;
   HoldingRegisters[4866] := 16#0000;
   HoldingRegisters[4867] := 16#0000;
   HoldingRegisters[4868] := 16#0000;
   HoldingRegisters[4869] := 16#0000;
   HoldingRegisters[4870] := 16#0000;
   HoldingRegisters[4871] := 16#0000;
   HoldingRegisters[4872] := 16#0000;
   HoldingRegisters[4873] := 16#0000;
   HoldingRegisters[4874] := 16#0000;
   HoldingRegisters[4875] := 16#0000;
   HoldingRegisters[4876] := 16#0000;
   HoldingRegisters[4877] := 16#0000;
   HoldingRegisters[4878] := 16#0000;
   HoldingRegisters[4879] := 16#0000;
   HoldingRegisters[4880] := 16#0000;
   HoldingRegisters[4881] := 16#0000;
   HoldingRegisters[4882] := 16#0000;
   HoldingRegisters[4883] := 16#0000;
   HoldingRegisters[4884] := 16#0000;
   HoldingRegisters[4885] := 16#0000;
   HoldingRegisters[4886] := 16#0000;
   HoldingRegisters[4887] := 16#0000;
   HoldingRegisters[4888] := 16#0000;
   HoldingRegisters[4889] := 16#0000;
   HoldingRegisters[4890] := 16#0000;
   HoldingRegisters[4891] := 16#0000;
   HoldingRegisters[4892] := 16#0000;
   HoldingRegisters[4893] := 16#0000;
   HoldingRegisters[4894] := 16#0000;
   HoldingRegisters[4895] := 16#0000;
   HoldingRegisters[4896] := 16#0000;
   HoldingRegisters[4897] := 16#0000;
   HoldingRegisters[4898] := 16#0000;
   HoldingRegisters[4899] := 16#0000;
   HoldingRegisters[4900] := 16#0000;
   HoldingRegisters[4901] := 16#0000;
   HoldingRegisters[4902] := 16#0000;
   HoldingRegisters[4903] := 16#0000;
   HoldingRegisters[4904] := 16#0000;
   HoldingRegisters[4905] := 16#0000;
   HoldingRegisters[4906] := 16#0000;
   HoldingRegisters[4907] := 16#0000;
   HoldingRegisters[4908] := 16#0000;
   HoldingRegisters[4909] := 16#0000;
   HoldingRegisters[4910] := 16#0000;
   HoldingRegisters[4911] := 16#0000;
   HoldingRegisters[4912] := 16#0000;
   HoldingRegisters[4913] := 16#0000;
   HoldingRegisters[4914] := 16#0000;
   HoldingRegisters[4915] := 16#0000;
   HoldingRegisters[4916] := 16#0000;
   HoldingRegisters[4917] := 16#0000;
   HoldingRegisters[4918] := 16#0000;
   HoldingRegisters[4919] := 16#0000;
   HoldingRegisters[4920] := 16#0000;
   HoldingRegisters[4921] := 16#0000;
   HoldingRegisters[4922] := 16#0000;
   HoldingRegisters[4923] := 16#0000;
   HoldingRegisters[4924] := 16#0000;
   HoldingRegisters[4925] := 16#0000;
   HoldingRegisters[4926] := 16#0000;
   HoldingRegisters[4927] := 16#0000;
   HoldingRegisters[4928] := 16#0000;
   HoldingRegisters[4929] := 16#0000;
   HoldingRegisters[4930] := 16#0000;
   HoldingRegisters[4931] := 16#0000;
   HoldingRegisters[4932] := 16#0000;
   HoldingRegisters[4933] := 16#0000;
   HoldingRegisters[4934] := 16#0000;
   HoldingRegisters[4935] := 16#0000;
   HoldingRegisters[4936] := 16#0000;
   HoldingRegisters[4937] := 16#0000;
   HoldingRegisters[4938] := 16#0000;
   HoldingRegisters[4939] := 16#0000;
   HoldingRegisters[4940] := 16#0000;
   HoldingRegisters[4941] := 16#0000;
   HoldingRegisters[4942] := 16#0000;
   HoldingRegisters[4943] := 16#0000;
   HoldingRegisters[4944] := 16#0000;
   HoldingRegisters[4945] := 16#0000;
   HoldingRegisters[4946] := 16#0000;
   HoldingRegisters[4947] := 16#0000;
   HoldingRegisters[4948] := 16#0000;
   HoldingRegisters[4949] := 16#0000;
   HoldingRegisters[4950] := 16#0000;
   HoldingRegisters[4951] := 16#0000;
   HoldingRegisters[4952] := 16#0000;
   HoldingRegisters[4953] := 16#0000;
   HoldingRegisters[4954] := 16#0000;
   HoldingRegisters[4955] := 16#0000;
   HoldingRegisters[4956] := 16#0000;
   HoldingRegisters[4957] := 16#0000;
   HoldingRegisters[4958] := 16#0000;
   HoldingRegisters[4959] := 16#0000;
   HoldingRegisters[4960] := 16#0000;
   HoldingRegisters[4961] := 16#0000;
   HoldingRegisters[4962] := 16#0000;
   HoldingRegisters[4963] := 16#0000;
   HoldingRegisters[4964] := 16#0000;
   HoldingRegisters[4965] := 16#0000;
   HoldingRegisters[4966] := 16#0000;
   HoldingRegisters[4967] := 16#0000;
   HoldingRegisters[4968] := 16#0000;
   HoldingRegisters[4969] := 16#0000;
   HoldingRegisters[4970] := 16#0000;
   HoldingRegisters[4971] := 16#0000;
   HoldingRegisters[4972] := 16#0000;
   HoldingRegisters[4973] := 16#0000;
   HoldingRegisters[4974] := 16#0000;
   HoldingRegisters[4975] := 16#0000;
   HoldingRegisters[4976] := 16#0000;
   HoldingRegisters[4977] := 16#0000;
   HoldingRegisters[4978] := 16#0000;
   HoldingRegisters[4979] := 16#0000;
   HoldingRegisters[4980] := 16#0000;
   HoldingRegisters[4981] := 16#0000;
   HoldingRegisters[4982] := 16#0000;
   HoldingRegisters[4983] := 16#0000;
   HoldingRegisters[4984] := 16#0000;
   HoldingRegisters[4985] := 16#0000;
   HoldingRegisters[4986] := 16#0000;
   HoldingRegisters[4987] := 16#0000;
   HoldingRegisters[4988] := 16#0000;
   HoldingRegisters[4989] := 16#0000;
   HoldingRegisters[4990] := 16#0000;
   HoldingRegisters[4991] := 16#0000;
   HoldingRegisters[4992] := 16#0000;
   HoldingRegisters[4993] := 16#0000;
   HoldingRegisters[4994] := 16#0000;
   HoldingRegisters[4995] := 16#0000;
   HoldingRegisters[4996] := 16#0000;
   HoldingRegisters[4997] := 16#0000;
   HoldingRegisters[4998] := 16#0000;
   HoldingRegisters[4999] := 16#0000;
END_DATA_BLOCK

DATA_BLOCK "OpcModel"   // DB4
{ S7_Optimized_Access := 'TRUE' }
VERSION : 0.1
   VAR
      FinalMaterial : String := 'PWT3021150020230526';
      MachineMode : Bool := TRUE;
      PlcReady : Bool := TRUE;
      Result : Int := 0;
      OffsetAngle : Real := 0.0;
      OffsetAngleMES : Real := 0.02;
      TestDone : Bool := FALSE;
      Control : Struct
         State : Int;
         Next : Bool;
         Recv : Struct
            Result : Int;
            OffsetAngle : Real;
            TestDone : Bool;
         END_STRUCT;
      END_STRUCT;
   END_VAR
BEGIN
END_DATA_BLOCK

DATA_BLOCK "Timer"   // DB5
{ S7_Optimized_Access := 'TRUE' }
VERSION : 0.1
   VAR
      DelayNextEDS : Int;
   END_VAR
BEGIN
END_DATA_BLOCK

// folder: (top level)

ORGANIZATION_BLOCK "Main"   // OB1, SCL, ProgramCycle
TITLE = "Main Program Sweep (Cycle)"
{ S7_Optimized_Access := 'TRUE' }
VERSION : 0.1
   VAR_INPUT
      Initial_Call : Bool;   // Initial call of this OB
      Remanence : Bool;   // =True, if remanent data are available
   END_VAR
BEGIN

   IF "Bit1s" THEN
       "SystemTick"();
       "Bit1s" := FALSE;
   END_IF;

   "ModbusTcpServer"();
   "OpcStack"();
END_ORGANIZATION_BLOCK

ORGANIZATION_BLOCK "Cyclic interrupt 1s"   // OB30, SCL, CyclicInterrupt
{ S7_Optimized_Access := 'TRUE' }
VERSION : 0.1
   VAR_INPUT
      Initial_Call : Bool;   // Initial call of this OB
      Event_Count : Int;   // Events discarded
   END_VAR
BEGIN
   "Bit1s" := true;
END_ORGANIZATION_BLOCK

ORGANIZATION_BLOCK "Startup"   // OB100, SCL, Startup
TITLE = "Complete Restart"
{ S7_Optimized_Access := 'TRUE' }
VERSION : 0.1
   VAR_INPUT
      LostRetentive : Bool;   // True if retentive data are lost
      LostRTC : Bool;   // True if date and time are lost
   END_VAR
BEGIN
END_ORGANIZATION_BLOCK

// folder: Sections

FUNCTION "ModbusTcpServer" : Void   // FC1, SCL
{ S7_Optimized_Access := 'TRUE' }
VERSION : 0.1
BEGIN


   "MB_SERVER_DB"(DISCONNECT:="ModbusModel".Disconnect,
                  NDR=>"ModbusModel"."NDR",
                  DR=>"ModbusModel".DR,
                  ERROR=>"ModbusModel".Error,
                  STATUS=>"ModbusModel".Status,
                  MB_HOLD_REG:="ModbusModel".HoldingRegisters,
                  CONNECT:="ModbusModel".Connect);

   (*Listen*)
   IF "ModbusModel".DR THEN
       "ModbusModel".DR := 0;
   ELSE
       ;
   END_IF;
END_FUNCTION

FUNCTION "OpcStack" : Void   // FC2, SCL
{ S7_Optimized_Access := 'TRUE' }
VERSION : 0.1
BEGIN

   case "OpcModel".Control.State OF
       0:
           "OpcModel".PlcReady := TRUE;
           //"OpcModel".FinalMaterial := 'PWT3021150020230526';
           "OpcModel".Control.State := "OpcModel".Control.State + 1;
       1:
           if "OpcModel".Result > 0 THEN
               "OpcModel".PlcReady := FALSE;

               // Next
               "Timer".DelayNextEDS := 10;
               "OpcModel".Control.State := "OpcModel".Control.State + 1;
           END_IF;
       2:
           if "Timer".DelayNextEDS = 0 THEN
               "OpcModel".Control.Next := true;
           END_IF;
           if "OpcModel".TestDone OR "OpcModel".Control.Next THEN
               // Save result here
               "OpcModel".Control.Recv.Result := "OpcModel".Result;
               "OpcModel".Control.Recv.OffsetAngle := "OpcModel".OffsetAngle;
               "OpcModel".Control.Recv.TestDone := "OpcModel".TestDone;

               "OpcModel".Result := 0;
               "OpcModel".OffsetAngle := 0.0;
               "OpcModel".TestDone := FALSE;
               // Next
               "OpcModel".Control.Next := false;
               "OpcModel".Control.State := "OpcModel".Control.State + 1;
           END_IF;
       ELSE
           "OpcModel".Control.State := 0;
   END_CASE;
END_FUNCTION

FUNCTION "SystemTick" : Void   // FC3, SCL
{ S7_Optimized_Access := 'TRUE' }
VERSION : 0.1
BEGIN

   IF "Timer".DelayNextEDS > 0 THEN
       "Timer".DelayNextEDS := "Timer".DelayNextEDS - 1;
   ELSE
       "Timer".DelayNextEDS := 0;
   END_IF;
END_FUNCTION